FUNCTION_BLOCK ValueObjectUDINT EXTENDS ValueObject
  VAR
    lValue : UDINT := 0;
    lOverrideValue : UDINT;
  END_VAR

            
          

METHOD configure
  VAR_INPUT
    executeContext : POINTER TO ExecuteContext;
  END_VAR
                  IF (executeContext^.configureUDINT(cTokenValue,lValue,FALSE,THIS)) THEN
	RETURN;
END_IF

IF (executeContext^.configureUDINT(cTokenOverrideValue,lOverrideValue,FALSE,THIS)) THEN
	RETURN;
END_IF

SUPER^.configure(executeContext);

                
END_METHOD

METHOD describe
  VAR_INPUT
    executeContext : POINTER TO ExecuteContext;
  END_VAR
                  SUPER^.describe(executeContext);

IF (executeContext^.matchOption(cExecuteOptionSyntax)) THEN
	executeContext^.describeSyntaxConfigurable(lStyle,cTokenValue,cDataTypeUDINT,cEnumTypeNone,lUnits,cDescriptionValue);
	executeContext^.describeSyntaxConfigurable(cValueStyleParameter,cTokenOverrideValue,cDataTypeUDINT,cEnumTypeNone,lUnits,cDescriptionOverrideValue);

	RETURN;
END_IF

IF (executeContext^.matchOption(cExecuteOptionParameter)) THEN
	executeContext^.describeParameter(lStyle,lIdentity,cTokenValue,gTypeHandler.getTokenForUDINT(lValue),cDataTypeUDINT,cEnumTypeNone,lUnits,cDescriptionValue);
	executeContext^.describeParameter(cValueStyleParameter,lIdentity,cTokenOverrideValue,gTypeHandler.getTokenForUDINT(lOverrideValue),cDataTypeUDINT,cEnumTypeNone,lUnits,cDescriptionOverrideValue);
		
	RETURN;
END_IF

executeContext^.appendTokenPair(cTokenValue,gTypeHandler.getTokenForUDINT(lValue),FALSE,TRUE);
executeContext^.appendTokenPair(cTokenOverrideValue,gTypeHandler.getTokenForUDINT(lOverrideValue),FALSE,TRUE);



                
END_METHOD

METHOD operator
                  IF (lOverride) THEN
	lValue := lOverrideValue;
END_IF


                
END_METHOD

PROPERTY OverrideValue : UDINT
GET
                    OverrideValue := lOverrideValue;
                  
END_GET
SET
                    lOverrideValue := OverrideValue;
                  
END_SET
END_PROPERTY

PROPERTY TypeToken : t_medium_string
GET
                    TypeToken := 'ValObjUDINT';
                  
END_GET
END_PROPERTY

(* {attribute 'monitoring' := 'call'} *)
PROPERTY Value : UDINT
GET
                    Value := lValue;
                  
END_GET
SET
                    lValue := Value;
                  
END_SET
END_PROPERTY
END_FUNCTION_BLOCK

FUNCTION_BLOCK ValueReferenceUDINT EXTENDS ValueReference
  VAR
    lValue : REFERENCE TO UDINT;
  END_VAR

            
          

METHOD configure
  VAR_INPUT
    executeContext : POINTER TO ExecuteContext;
  END_VAR
                  IF (executeContext^.configureUDINT(cTokenValue,lValue,FALSE,THIS)) THEN
	RETURN;
END_IF

SUPER^.configure(executeContext);


                
END_METHOD

METHOD describe
  VAR_INPUT
    executeContext : POINTER TO ExecuteContext;
  END_VAR
                  IF (executeContext^.matchOption(cExecuteOptionParameter)) THEN
	executeContext^.describeParameter(lStyle,lIdentity,cTokenValue,gTypeHandler.getTokenForUDINT(lValue),cDataTypeUDINT,cEnumTypeNone,lUnits,cDescriptionValue);
	RETURN;
END_IF

SUPER^.describe(executeContext);

IF (executeContext^.matchOption(cExecuteOptionSyntax)) THEN
	executeContext^.describeSyntaxConfigurable(lStyle,cTokenValue,cDataTypeUDINT,cEnumTypeNone,lUnits,cDescriptionValue);
	RETURN;
END_IF

executeContext^.appendTokenPair(cTokenValue,gTypeHandler.getTokenForUDINT(lValue),FALSE,TRUE);





                
END_METHOD

METHOD initializeValueReference
  VAR_INPUT
    value : REFERENCE TO UDINT;
    p : POINTER TO t_particle_nop;
    _name : t_medium_string;
    description : t_long_string;
    units : t_token_string;
    style : t_value_style;
  END_VAR
                  lValue REF= value;
Name := _name;
Description := description;
lUnits := units;
lStyle := style;

IF (p<>0) THEN
	p^.registerNonOperational(THIS);
END_IF

                
END_METHOD

PROPERTY TypeToken : t_medium_string
GET
                    TypeToken := 'ValRefUDINT';
                  
END_GET
END_PROPERTY

PROPERTY Value : UDINT
GET
                    Value := lValue;
                  
END_GET
SET
                    lValue := Value;
                  
END_SET
END_PROPERTY
END_FUNCTION_BLOCK

FUNCTION_BLOCK ValueObjectUINTInputReferenceUINT EXTENDS ValueObjectUINT
  VAR
    lInputReference : REFERENCE TO UINT;
  END_VAR

            
          

METHOD initialize
                  IF (NOT(__ISVALIDREF(lInputReference))) THEN
	gCodeErrorHandler(pMessage:=CONCAT('null reference in ',lIdentity));
END_IF

SUPER^.initialize();

                
END_METHOD

METHOD operator
                  lValue := lInputReference;

SUPER^.operator();

                
END_METHOD

PROPERTY InputReference : REFERENCE TO UINT
SET
                    lInputReference REF= InputReference;


                  
END_SET
END_PROPERTY
END_FUNCTION_BLOCK

FUNCTION_BLOCK ValueObjectUINTOutputReferenceUINT EXTENDS ValueObjectUINT
  VAR
    lOutputReference : REFERENCE TO UINT;
  END_VAR

            
          

METHOD initialize
                  IF (NOT(__ISVALIDREF(lOutputReference))) THEN
	gCodeErrorHandler(pMessage:=CONCAT('null reference in ',lIdentity));
END_IF

SUPER^.initialize();

                
END_METHOD

METHOD operator
                  SUPER^.operator();

lOutputReference := lValue;
                
END_METHOD

PROPERTY OutputReference : REFERENCE TO UINT
SET
                    lOutputReference ref= OutputReference;
                  
END_SET
END_PROPERTY
END_FUNCTION_BLOCK

FUNCTION_BLOCK ValueObjectUINT EXTENDS ValueObject
  VAR
    lValue : UINT := 0;
    lOverrideValue : UINT := 0;
  END_VAR

            
          

METHOD configure
  VAR_INPUT
    executeContext : POINTER TO ExecuteContext;
  END_VAR
                  IF (executeContext^.configureUINT(cTokenValue,lValue,FALSE,THIS)) THEN
	RETURN;
END_IF

IF (executeContext^.configureUINT(cTokenOverrideValue,lOverrideValue,FALSE,THIS)) THEN
	RETURN;
END_IF

SUPER^.configure(executeContext);

                
END_METHOD

METHOD describe
  VAR_INPUT
    executeContext : POINTER TO ExecuteContext;
  END_VAR
                  SUPER^.describe(executeContext);

IF (executeContext^.matchOption(cExecuteOptionSyntax)) THEN
	executeContext^.describeSyntaxConfigurable(lStyle,cTokenValue,cDataTypeUINT,cEnumTypeNone,lUnits,cDescriptionValue);
	executeContext^.describeSyntaxConfigurable(cValueStyleParameter,cTokenOverrideValue,cDataTypeUINT,cEnumTypeNone,lUnits,cDescriptionOverrideValue);

	RETURN;
END_IF

IF (executeContext^.matchOption(cExecuteOptionParameter)) THEN
	executeContext^.describeParameter(lStyle,lIdentity,cTokenValue,gTypeHandler.getTokenForUINT(lValue),cDataTypeUINT,cEnumTypeNone,lUnits,cDescriptionValue);
	executeContext^.describeParameter(cValueStyleParameter,lIdentity,cTokenOverrideValue,gTypeHandler.getTokenForUINT(lOverrideValue),cDataTypeUINT,cEnumTypeNone,lUnits,cDescriptionOverrideValue);
		
	RETURN;
END_IF

executeContext^.appendTokenPair(cTokenValue,gTypeHandler.getTokenForUINT(lValue),FALSE,TRUE);
executeContext^.appendTokenPair(cTokenOverrideValue,gTypeHandler.getTokenForUINT(lOverrideValue),FALSE,TRUE);




                
END_METHOD

METHOD operator
                  IF (lOverride) THEN
	lValue := lOverrideValue;
END_IF

                
END_METHOD

PROPERTY OverrideValue : UINT
GET
                    OverrideValue := lOverrideValue;
                  
END_GET
SET
                    lOverrideValue := OverrideValue;
                  
END_SET
END_PROPERTY

PROPERTY TypeToken : t_medium_string
GET
                    TypeToken := 'ValObjUINT';
                  
END_GET
END_PROPERTY

PROPERTY Value : UINT
GET
                    Value := lValue;
                  
END_GET
SET
                    lValue := Value;
                  
END_SET
END_PROPERTY

PROPERTY ValueReference : REFERENCE TO UINT
GET
                    ValueReference REF= lValue;

                  
END_GET
END_PROPERTY
END_FUNCTION_BLOCK

FUNCTION_BLOCK ValueReferencePersistentUINT EXTENDS ValueReference
  VAR
    lValue : REFERENCE TO t_persistent_uint;
  END_VAR

            
          

METHOD describe
  VAR_INPUT
    executeContext : POINTER TO ExecuteContext;
  END_VAR
                  IF (executeContext^.matchOption(cExecuteOptionParameter)) THEN
	executeContext^.describeParameter(lStyle,lIdentity,cTokenValue,gTypeHandler.getTokenForUINT(lValue.Value),cDataTypeUINT,cEnumTypeNone,lUnits,cDescriptionValue);	
	RETURN;
END_IF

SUPER^.describe(executeContext);

IF (executeContext^.matchOption(cExecuteOptionSyntax)) THEN
	executeContext^.describeSyntaxConfigurable(lStyle,cTokenValue,cDataTypeUINT,cEnumTypeNone,lUnits,cDescriptionValue);
	RETURN;
END_IF

executeContext^.appendTokenPair(cTokenValue,gTypeHandler.getTokenForUINT(lValue.Value),FALSE,TRUE);

                
END_METHOD

METHOD configure
  VAR_INPUT
    executeContext : POINTER TO ExecuteContext;
  END_VAR
  VAR
    value : UINT;
  END_VAR
                  IF (executeContext^.configureUINT(cTokenValue,value,FALSE,THIS)) THEN
	lValue.Value := value;
	RETURN;
END_IF

SUPER^.configure(executeContext);

                
END_METHOD

METHOD initializeValueReference
  VAR_INPUT
    value : REFERENCE TO t_persistent_uint;
    p : POINTER TO t_particle_nop;
    _name : t_medium_string;
    description : t_long_string;
    units : t_token_string;
    style : t_value_style;
  END_VAR
                  lValue REF= value;
Name := _name;
Description := description;
lUnits := units;
lStyle := style;

IF (p<>0) THEN
	p^.registerNonOperational(THIS);
END_IF

                
END_METHOD

PROPERTY TypeToken : t_medium_string
GET
                    TypeToken := 'ValRefPersUINT';
                  
END_GET
END_PROPERTY

PROPERTY Value : UINT
GET
                    Value := lValue.Value;
                  
END_GET
SET
                    lValue.Value := Value;
                  
END_SET
END_PROPERTY
END_FUNCTION_BLOCK

FUNCTION_BLOCK ValueReferenceUINT EXTENDS ValueReference
  VAR
    lValue : REFERENCE TO UINT;
  END_VAR

            
          

METHOD configure
  VAR_INPUT
    executeContext : POINTER TO ExecuteContext;
  END_VAR
                  IF (executeContext^.configureUINT(cTokenValue,lValue,FALSE,THIS)) THEN
	RETURN;
END_IF

SUPER^.configure(executeContext);


                
END_METHOD

METHOD initializeValueReference
  VAR_INPUT
    value : REFERENCE TO UINT;
    p : POINTER TO t_particle_nop;
    _name : t_medium_string;
    description : t_long_string;
    units : t_token_string;
    style : t_value_style;
  END_VAR
                  lValue REF= value;
Name := _name;
Description := description;
lUnits := units;
lStyle := style;

IF (p<>0) THEN
	p^.registerNonOperational(THIS);
END_IF

                
END_METHOD

METHOD describe
  VAR_INPUT
    executeContext : POINTER TO ExecuteContext;
  END_VAR
                  IF (executeContext^.matchOption(cExecuteOptionParameter)) THEN
	executeContext^.describeParameter(lStyle,lIdentity,cTokenValue,gTypeHandler.getTokenForUINT(lValue),cDataTypeUINT,cEnumTypeNone,lUnits,cDescriptionValue);
	RETURN;
END_IF

SUPER^.describe(executeContext);

IF (executeContext^.matchOption(cExecuteOptionSyntax)) THEN
	executeContext^.describeSyntaxConfigurable(lStyle,cTokenValue,cDataTypeUINT,cEnumTypeNone,lUnits,cDescriptionValue);
	RETURN;
END_IF

executeContext^.appendTokenPair(cTokenValue,gTypeHandler.getTokenForUINT(lValue),FALSE,TRUE);



                
END_METHOD

PROPERTY TypeToken : t_medium_string
GET
                    TypeToken := 'ValRefUINT';
                  
END_GET
END_PROPERTY

PROPERTY Value : UINT
GET
                    Value := lValue;
                  
END_GET
SET
                    lValue := Value;
                  
END_SET
END_PROPERTY
END_FUNCTION_BLOCK

FUNCTION_BLOCK ValueObjectULINTInputReferenceULINT EXTENDS ValueObjectULINT
  VAR
    lInputReference : REFERENCE TO ULINT;
  END_VAR

            
          

METHOD initialize
                  IF (NOT(__ISVALIDREF(lInputReference))) THEN
	gCodeErrorHandler(pMessage:=CONCAT('null reference in ',lIdentity));
END_IF

SUPER^.initialize();

                
END_METHOD

METHOD operator
                  lValue := lInputReference;

SUPER^.operator();

                
END_METHOD

PROPERTY InputReference : REFERENCE TO ULINT
SET
                    lInputReference REF= InputReference;


                  
END_SET
END_PROPERTY
END_FUNCTION_BLOCK

FUNCTION_BLOCK ValueObjectULINT EXTENDS ValueObject
  VAR
    lValue : ULINT := 0;
    lOverrideValue : ULINT;
  END_VAR

            
          

METHOD configure
  VAR_INPUT
    executeContext : POINTER TO ExecuteContext;
  END_VAR
                  IF (executeContext^.configureULINT(cTokenValue,lValue,FALSE,THIS)) THEN
	RETURN;
END_IF

IF (executeContext^.configureULINT(cTokenOverrideValue,lOverrideValue,FALSE,THIS)) THEN
	RETURN;
END_IF

SUPER^.configure(executeContext);


                
END_METHOD

METHOD describe
  VAR_INPUT
    executeContext : POINTER TO ExecuteContext;
  END_VAR
                  SUPER^.describe(executeContext);

IF (executeContext^.matchOption(cExecuteOptionSyntax)) THEN
	executeContext^.describeSyntaxConfigurable(lStyle,cTokenValue,cDataTypeULINT,cEnumTypeNone,lUnits,cDescriptionValue);
	executeContext^.describeSyntaxConfigurable(cValueStyleParameter,cTokenOverrideValue,cDataTypeULINT,cEnumTypeNone,lUnits,cDescriptionOverrideValue);
	
	RETURN;
END_IF

IF (executeContext^.matchOption(cExecuteOptionParameter)) THEN
	executeContext^.describeParameter(lStyle,lIdentity,cTokenValue,gTypeHandler.getTokenForULINT(lValue),cDataTypeULINT,cEnumTypeNone,lUnits,cDescriptionValue);
	executeContext^.describeParameter(cValueStyleParameter,lIdentity,cTokenOverrideValue,gTypeHandler.getTokenForULINT(lOverrideValue),cDataTypeULINT,cEnumTypeNone,lUnits,cDescriptionOverrideValue);
		
	RETURN;
END_IF

executeContext^.appendTokenPair(cTokenValue,gTypeHandler.getTokenForULINT(lValue),FALSE,TRUE);
executeContext^.appendTokenPair(cTokenOverrideValue,gTypeHandler.getTokenForULINT(lOverrideValue),FALSE,TRUE);



                
END_METHOD

METHOD operator
                  IF (lOverride) THEN
	lValue := lOverrideValue;
END_IF


                
END_METHOD

PROPERTY OverrideValue : ULINT
GET
                    OverrideValue := lOverrideValue;
                  
END_GET
SET
                    lOverrideValue := OverrideValue;
                  
END_SET
END_PROPERTY

PROPERTY TypeToken : t_medium_string
GET
                    TypeToken := 'ValObjULINT';
                  
END_GET
END_PROPERTY

PROPERTY Value : ULINT
GET
                    Value := lValue;
                  
END_GET
SET
                    lValue := Value;
                  
END_SET
END_PROPERTY
END_FUNCTION_BLOCK

FUNCTION_BLOCK ValueReferenceULINT EXTENDS ValueReference
  VAR
    lValue : REFERENCE TO ULINT;
  END_VAR

            
          

METHOD configure
  VAR_INPUT
    executeContext : POINTER TO ExecuteContext;
  END_VAR
                  IF (executeContext^.configureULINT(cTokenValue,lValue,FALSE,THIS)) THEN
	RETURN;
END_IF

SUPER^.configure(executeContext);



                
END_METHOD

METHOD describe
  VAR_INPUT
    executeContext : POINTER TO ExecuteContext;
  END_VAR
                  IF (executeContext^.matchOption(cExecuteOptionParameter)) THEN
	executeContext^.describeParameter(lStyle,lIdentity,cTokenValue,gTypeHandler.getTokenForULINT(lValue),cDataTypeULINT,cEnumTypeNone,lUnits,cDescriptionValue);
	RETURN;
END_IF

SUPER^.describe(executeContext);

IF (executeContext^.matchOption(cExecuteOptionSyntax)) THEN
	executeContext^.describeSyntaxConfigurable(lStyle,cTokenValue,cDataTypeULINT,cEnumTypeNone,lUnits,cDescriptionValue);
	RETURN;
END_IF

executeContext^.appendTokenPair(cTokenValue,gTypeHandler.getTokenForULINT(lValue),FALSE,TRUE);



                
END_METHOD

METHOD initializeValueReference
  VAR_INPUT
    value : REFERENCE TO ULINT;
    p : POINTER TO t_particle_nop;
    _name : t_medium_string;
    description : t_long_string;
    units : t_token_string;
    style : t_value_style;
  END_VAR
                  lValue REF= value;
Name := _name;
Description := description;
lUnits := units;
lStyle := style;

IF (p<>0) THEN
	p^.registerNonOperational(THIS);
END_IF

                
END_METHOD

PROPERTY TypeToken : t_medium_string
GET
                    TypeToken := 'ValRefULINT';
                  
END_GET
END_PROPERTY

PROPERTY Value : ULINT
GET
                    Value := lValue;
                  
END_GET
SET
                    lValue := Value;
                  
END_SET
END_PROPERTY
END_FUNCTION_BLOCK

FUNCTION_BLOCK ValueObjectUSINTInputReferenceUSINT EXTENDS ValueObjectUSINT
  VAR
    lInputReference : REFERENCE TO USINT;
  END_VAR

            
          

METHOD initialize
                  IF (NOT(__ISVALIDREF(lInputReference))) THEN
	gCodeErrorHandler(pMessage:=CONCAT('null reference in ',lIdentity));
END_IF

SUPER^.initialize();

                
END_METHOD

METHOD operator
                  lValue := lInputReference;

SUPER^.operator();

                
END_METHOD

PROPERTY InputReference : REFERENCE TO USINT
SET
                    lInputReference REF= InputReference;


                  
END_SET
END_PROPERTY
END_FUNCTION_BLOCK

FUNCTION_BLOCK ValueObjectUSINTInputUSINT EXTENDS ValueObjectUSINT
  VAR
    lInput : USINT;
  END_VAR

            
          

METHOD operator
                  lValue := lInput;

SUPER^.operator();

                
END_METHOD

PROPERTY Input : USINT
SET
                    lInput := Input;
operator();

                  
END_SET
END_PROPERTY
END_FUNCTION_BLOCK

FUNCTION_BLOCK ValueObjectUSINTOutputReferenceUSINT EXTENDS ValueObjectUSINT
  VAR
    lOutputReference : REFERENCE TO USINT;
  END_VAR

            
          

METHOD initialize
                  IF (NOT(__ISVALIDREF(lOutputReference))) THEN
	gCodeErrorHandler(pMessage:=CONCAT('null reference in ',lIdentity));
END_IF

SUPER^.initialize();

                
END_METHOD

METHOD operator
                  SUPER^.operator();

lOutputReference := lValue;

                
END_METHOD

PROPERTY OutputReference : REFERENCE TO USINT
SET
                    lOutputReference ref= OutputReference;
                  
END_SET
END_PROPERTY
END_FUNCTION_BLOCK

FUNCTION_BLOCK ValueObjectUSINT EXTENDS ValueObject
  VAR
    lValue : USINT := 0;
    lOverrideValue : USINT := 0;
  END_VAR

            
          

METHOD configure
  VAR_INPUT
    executeContext : POINTER TO ExecuteContext;
  END_VAR
                  IF (executeContext^.configureUSINT(cTokenValue,lValue,FALSE,THIS)) THEN
	RETURN;
END_IF

IF (executeContext^.configureUSINT(cTokenOverrideValue,lOverrideValue,FALSE,THIS)) THEN
	RETURN;
END_IF

SUPER^.configure(executeContext);

                
END_METHOD

METHOD describe
  VAR_INPUT
    executeContext : POINTER TO ExecuteContext;
  END_VAR
                  SUPER^.describe(executeContext);

IF (executeContext^.matchOption(cExecuteOptionSyntax)) THEN
	executeContext^.describeSyntaxConfigurable(lStyle,cTokenValue,cDataTypeUSINT,cEnumTypeNone,lUnits,cDescriptionValue);
	executeContext^.describeSyntaxConfigurable(cValueStyleParameter,cTokenOverrideValue,cDataTypeUSINT,cEnumTypeNone,lUnits,cDescriptionOverrideValue);

	RETURN;
END_IF

IF (executeContext^.matchOption(cExecuteOptionParameter)) THEN
	executeContext^.describeParameter(lStyle,lIdentity,cTokenValue,gTypeHandler.getTokenForUSINT(lValue),cDataTypeUSINT,cEnumTypeNone,lUnits,cDescriptionValue);
	executeContext^.describeParameter(cValueStyleParameter,lIdentity,cTokenOverrideValue,gTypeHandler.getTokenForUSINT(lOverrideValue),cDataTypeUSINT,cEnumTypeNone,lUnits,cDescriptionOverrideValue);
	
	RETURN;
END_IF

executeContext^.appendTokenPair(cTokenValue,gTypeHandler.getTokenForUSINT(lValue),FALSE,TRUE);
executeContext^.appendTokenPair(cTokenOverrideValue,gTypeHandler.getTokenForUSINT(lOverrideValue),FALSE,TRUE);

                
END_METHOD

METHOD operator
                  IF (lOverride) THEN
	lValue := lOverrideValue;
END_IF


                
END_METHOD

PROPERTY OverrideValue : USINT
GET
                    OverrideValue := lOverrideValue;
                  
END_GET
SET
                    lOverrideValue := OverrideValue;
                  
END_SET
END_PROPERTY

PROPERTY TypeToken : t_medium_string
GET
                    TypeToken := 'ValObjUSINT';
                  
END_GET
END_PROPERTY

(* {attribute 'monitoring' := 'call'} *)
PROPERTY Value : USINT
GET
                    Value := lValue;
                  
END_GET
SET
                    lValue := Value;
                  
END_SET
END_PROPERTY
END_FUNCTION_BLOCK

FUNCTION_BLOCK ValueReferenceUSINT EXTENDS ValueReference
  VAR
    lValue : REFERENCE TO USINT;
  END_VAR

            
          

METHOD configure
  VAR_INPUT
    executeContext : POINTER TO ExecuteContext;
  END_VAR
                  IF (executeContext^.configureUSINT(cTokenValue,lValue,FALSE,THIS)) THEN
	RETURN;
END_IF

SUPER^.configure(executeContext);

                
END_METHOD

METHOD describe
  VAR_INPUT
    executeContext : POINTER TO ExecuteContext;
  END_VAR
                  IF (executeContext^.matchOption(cExecuteOptionParameter)) THEN
	executeContext^.describeParameter(lStyle,lIdentity,cTokenValue,gTypeHandler.getTokenForUSINT(lValue),cDataTypeUSINT,cEnumTypeNone,lUnits,cDescriptionValue);
	RETURN;
END_IF

SUPER^.describe(executeContext);

IF (executeContext^.matchOption(cExecuteOptionSyntax)) THEN
	executeContext^.describeSyntaxConfigurable(lStyle,cTokenValue,cDataTypeUSINT,cEnumTypeNone,lUnits,cDescriptionValue);
	RETURN;
END_IF

executeContext^.appendTokenPair(cTokenValue,gTypeHandler.getTokenForUSINT(lValue),FALSE,TRUE);



                
END_METHOD

METHOD initializeValueReference
  VAR_INPUT
    value : REFERENCE TO USINT;
    p : POINTER TO t_particle_nop;
    _name : t_medium_string;
    description : t_long_string;
    units : t_token_string;
    style : t_value_style;
  END_VAR
                  lValue REF= value;
Name := _name;
Description := description;
lUnits := units;
lStyle := style;

IF (p<>0) THEN
	p^.registerNonOperational(THIS);
END_IF

                
END_METHOD

PROPERTY TypeToken : t_medium_string
GET
                    TypeToken := 'ValRefUSINT';
                  
END_GET
END_PROPERTY

PROPERTY Value : USINT
GET
                    Value := lValue;
                  
END_GET
SET
                    lValue := Value;
                  
END_SET
END_PROPERTY
END_FUNCTION_BLOCK

FUNCTION_BLOCK ValueObject EXTENDS Particle
  VAR
    lUnits : t_token_string;
    lOverride : BOOL := FALSE;
    lStyle : t_value_style := cValueStyleConfigurable;
  END_VAR

            
          

METHOD describe
  VAR_INPUT
    executeContext : POINTER TO ExecuteContext;
  END_VAR
                  SUPER^.describe(executeContext);

IF (executeContext^.matchOption(cExecuteOptionSyntax)) THEN
	executeContext^.describeSyntaxConfigurable(cValueStyleParameter,cTokenOverride,cDataTypeBool,cEnumTypeNone,lUnits,cDescriptionOverride);
	RETURN;
END_IF

IF (executeContext^.matchOption(cExecuteOptionParameter)) THEN
	executeContext^.describeParameter(cValueStyleParameter,lIdentity,cTokenOverride,gTypeHandler.getTokenForBool(lOverride),cDataTypeBool,cEnumTypeNone,lUnits,cDescriptionOverride);

	RETURN;
END_IF

executeContext^.appendTokenPair(cTokenOverride,gTypeHandler.getTokenForUSINT(BOOL_TO_USINT(lOverride)),FALSE,TRUE);


                
END_METHOD

METHOD initializeValueObject
  VAR_INPUT
    p : POINTER TO t_particle_nop;
    _name : t_medium_string;
    description : t_long_string;
    units : t_token_string;
    style : t_value_style;
  END_VAR
                  Name := _name;
Description := description;
lUnits := units;
lStyle := style;

IF (p=0) THEN
	gCodeErrorHandler(pMessage:='initializing value with null t_particle_nop');
	RETURN;
END_IF

p^.registerNonOperational(THIS);

                
END_METHOD

METHOD initializeValueObjectOp
  VAR_INPUT
    p : POINTER TO t_particle_op;
    _name : t_medium_string;
    description : t_long_string;
    units : t_token_string;
    style : t_value_style;
  END_VAR
                  Name := _name;
Description := description;
lUnits := units;
lStyle := style;

IF (p=0) THEN
	gCodeErrorHandler(pMessage:='initializing value with null t_particle_op');
	RETURN;
END_IF

p^.registerOperational(THIS);

                
END_METHOD

METHOD configure
  VAR_INPUT
    executeContext : POINTER TO ExecuteContext;
  END_VAR
                  IF (executeContext^.configureBool(cTokenOverride,lOverride,FALSE,THIS)) THEN
	RETURN;
END_IF

SUPER^.configure(executeContext);

                
END_METHOD

PROPERTY Override : BOOL
GET
                    Override := lOverride;
                  
END_GET
SET
                    lOverride := Override;
                  
END_SET
END_PROPERTY

PROPERTY TypeToken : t_medium_string
GET
                    TypeToken := 'ValueObject';
                  
END_GET
END_PROPERTY
END_FUNCTION_BLOCK

FUNCTION_BLOCK ValueReference EXTENDS Particle
  VAR
    lUnits : t_token_string;
    lStyle : t_value_style := cValueStyleConfigurable;
  END_VAR

            
          

PROPERTY TypeToken : t_medium_string
GET
                    TypeToken := 'ValueReference';
                  
END_GET
END_PROPERTY
END_FUNCTION_BLOCK

FUNCTION_BLOCK ExecuteCommand
  VAR
    lCommand : t_token_type;
    lOptions : t_options_list;
    lPairs : ARRAY[1..4] OF t_argument;
  END_VAR

            
          
END_FUNCTION_BLOCK

{attribute 'enable_dynamic_creation'}
FUNCTION_BLOCK ExecuteContext
  VAR CONSTANT
    cExecuteLimit : USINT := 2;
    cExecutionQueueMax : UINT := 4096;
    cParseMaxTokens : USINT := 32;
    cSkipCount : USINT := 5;
  END_VAR
  VAR
    lExecutionQueue : ARRAY[1..cExecutionQueueMax] OF t_execution_queue_item;  (* lSource: REFERENCE TO t_execute_source; *)
    lExecutionQueueCount : UINT;
    lExecutionQueueIndex : UINT;
    lRegisterDepth : USINT;
    lCurrentCommand : t_command_request;
    lExecuteReturn : t_execute_return := cExecuteReturnOK;
    lResponsePending : BOOL := FALSE;
    lError : BOOL := FALSE;
    lReportError : BOOL := FALSE;
    lWriteStream : t_stream;
    lEnableExecutor : BOOL := TRUE;
    lReadWrite : BOOL := FALSE;
    lPassCount : USINT;
    lPassLimit : USINT := cExecuteLimit;
    lSkipIndex : USINT := 0;
    lSkipCount : USINT := cSkipCount;
    lCommaPending : BOOL := FALSE;
    lWrappedResponse : BOOL := FALSE;
  END_VAR

            
          

METHOD configureDWORD : BOOL
  VAR_INPUT
    parameter : t_token_type;
    target : REFERENCE TO DWORD;
    required : BOOL;
    particle : POINTER TO t_particle;
  END_VAR
  VAR
    valueToken : t_token_string;
  END_VAR
                  configureDWORD := matchArgument(parameter,valueToken);

IF (NOT(configureDWORD)) THEN
	IF (required) THEN
		executeContextFail(THIS,cExecuteReturnMissingArgument,TRUE);		
	END_IF
	
	RETURN;
END_IF

IF (NOT(gTypeHandler.getDWORDFromToken(valueToken,target))) THEN
	executeContextFail(THIS,cExecuteReturnParseParameterError,TRUE);
	RETURN;
END_IF

gSystemServices.Executor.reportParameterUpdates(particle);

                
END_METHOD

METHOD describeSyntaxConfigurable
  VAR_INPUT
    style : t_value_style;
    parameter : t_token_type;
    dataType : t_data_type;
    enumType : t_enum_type;
    units : t_token_string;
    description : REFERENCE TO t_long_string;
  END_VAR
                  recordInitiator();

appendTokenPair(parameter,gTypeHandler.getTokenForDataType(dataType),TRUE,FALSE);

append(', "_metadata":');
recordInitiator();

appendPair('style',gTypeHandler.getTokenForEnum(cEnumTypeValueStyle,style),TRUE,FALSE);
appendPair('units',units,TRUE,TRUE);
appendPair('description',description,TRUE,TRUE);

IF (enumType<>cEnumTypeNone) THEN
	appendPair('enum',gTypeHandler.getStringForEnumOptions(enumType),FALSE,TRUE);
END_IF

recordTerminator();
recordTerminatorWithNewline();

                
END_METHOD

METHOD configureUSINT : BOOL
  VAR_INPUT
    parameter : t_token_type;
    target : REFERENCE TO USINT;
    required : BOOL;
    particle : POINTER TO t_particle;
  END_VAR
  VAR
    valueToken : t_token_string;
  END_VAR
                  configureUSINT := matchArgument(parameter,valueToken);

IF (NOT(configureUSINT)) THEN
	IF (required) THEN
		executeContextFail(THIS,cExecuteReturnMissingArgument,TRUE);		
	END_IF
	
	RETURN;
END_IF

IF (NOT(gTypeHandler.getUSINTFromToken(valueToken,target))) THEN
	executeContextFail(THIS,cExecuteReturnParseParameterError,TRUE);
	RETURN;
END_IF

gSystemServices.Executor.reportParameterUpdates(particle);

                
END_METHOD

METHOD recordInitiatorWithNewlineIndent
                  formatWithNewlineIndent();
lWriteStream.recordInitiator();

                
END_METHOD

METHOD formatWithNewlineIndent
                  IF (NOT(lWrappedResponse)) THEN
	lWriteStream.newline();
	lWriteStream.indent();
END_IF


                
END_METHOD

METHOD append
  VAR_INPUT
    str : STRING;
  END_VAR
                  lWriteStream.append(str);

                
END_METHOD

METHOD configureUINT : BOOL
  VAR_INPUT
    parameter : t_token_type;
    target : REFERENCE TO UINT;
    required : BOOL;
    particle : POINTER TO t_particle;
  END_VAR
  VAR
    valueToken : t_token_string;
  END_VAR
                  configureUINT := matchArgument(parameter,valueToken);

IF (NOT(configureUINT)) THEN
	IF (required) THEN
		executeContextFail(THIS,cExecuteReturnMissingArgument,TRUE);		
	END_IF
	
	RETURN;
END_IF

IF (NOT(gTypeHandler.getUINTFromToken(valueToken,target))) THEN
	executeContextFail(THIS,cExecuteReturnParseParameterError,TRUE);
	RETURN;
END_IF

gSystemServices.Executor.reportParameterUpdates(particle);

                
END_METHOD

METHOD configureMediumString : BOOL
  VAR_INPUT
    parameter : t_token_type;
    target : REFERENCE TO t_medium_string;
    required : BOOL;
    particle : POINTER TO t_particle;
  END_VAR
  VAR
    valueToken : t_token_string;
  END_VAR
                  configureMediumString := matchArgument(parameter,valueToken);

IF (NOT(configureMediumString)) THEN
	IF (required) THEN
		executeContextFail(THIS,cExecuteReturnMissingArgument,TRUE);		
	END_IF
	
	RETURN;
END_IF

target := valueToken;

gSystemServices.Executor.reportParameterUpdates(particle);

                
END_METHOD

METHOD configureUDINT : BOOL
  VAR_INPUT
    parameter : t_token_type;
    target : REFERENCE TO UDINT;
    required : BOOL;
    particle : POINTER TO t_particle;
  END_VAR
  VAR
    valueToken : t_token_string;
  END_VAR
                  configureUDINT := matchArgument(parameter,valueToken);

IF (NOT(configureUDINT)) THEN
	IF (required) THEN
		executeContextFail(THIS,cExecuteReturnMissingArgument,TRUE);		
	END_IF
	
	RETURN;
END_IF

IF (NOT(gTypeHandler.getUDINTFromToken(valueToken,target))) THEN
	executeContextFail(THIS,cExecuteReturnParseParameterError,TRUE);
	RETURN;
END_IF

gSystemServices.Executor.reportParameterUpdates(particle);


                
END_METHOD

METHOD configureReal : BOOL
  VAR_INPUT
    parameter : t_token_type;
    target : REFERENCE TO REAL;
    required : BOOL;
    particle : POINTER TO t_particle;
  END_VAR
  VAR
    valueToken : t_token_string;
  END_VAR
                  configureReal := matchArgument(parameter,valueToken);

IF (NOT(configureReal)) THEN
	IF (required) THEN
		executeContextFail(THIS,cExecuteReturnMissingArgument,TRUE);		
	END_IF
	
	RETURN;
END_IF

IF (NOT(gTypeHandler.getREALFromToken(valueToken,target))) THEN
	executeContextFail(THIS,cExecuteReturnParseParameterError,TRUE);
	RETURN;
END_IF

gSystemServices.Executor.reportParameterUpdates(particle);


                
END_METHOD

METHOD configurePercentage : BOOL
  VAR_INPUT
    parameter : t_token_type;
    target : REFERENCE TO t_percentage;
    required : BOOL;
    particle : POINTER TO t_particle;
  END_VAR
  VAR
    valueToken : t_token_string;
  END_VAR
                  configurePercentage := matchArgument(parameter,valueToken);

IF (NOT(configurePercentage)) THEN
	IF (required) THEN
		executeContextFail(THIS,cExecuteReturnMissingArgument,TRUE);		
	END_IF
	
	RETURN;
END_IF

IF (NOT(gTypeHandler.getPercentageFromToken(valueToken,target))) THEN
	executeContextFail(THIS,cExecuteReturnParseParameterError,TRUE);
	RETURN;
END_IF

gSystemServices.Executor.reportParameterUpdates(particle);


                
END_METHOD

METHOD configureEnum : BOOL
  VAR_INPUT
    enumType : t_enum_type;
    parameter : t_token_type;
    target : REFERENCE TO INT;
    required : BOOL;
    particle : POINTER TO t_particle;
  END_VAR
  VAR
    valueToken : t_token_string;
  END_VAR
                  configureEnum := matchArgument(parameter,valueToken);

IF (NOT(configureEnum)) THEN
	IF (required) THEN
		executeContextFail(THIS,cExecuteReturnMissingArgument,TRUE);		
	END_IF
	
	RETURN;
END_IF

IF (NOT(gTypeHandler.getEnumFromToken(enumType,valueToken,target))) THEN
	executeContextFail(THIS,cExecuteReturnParseParameterError,TRUE);
	RETURN;
END_IF

gSystemServices.Executor.reportParameterUpdates(particle);


                
END_METHOD

METHOD configureULINT : BOOL
  VAR_INPUT
    parameter : t_token_type;
    target : REFERENCE TO ULINT;
    required : BOOL;
    particle : POINTER TO t_particle;
  END_VAR
  VAR
    valueToken : t_token_string;
  END_VAR
                  configureULINT := matchArgument(parameter,valueToken);

IF (NOT(configureULINT)) THEN
	IF (required) THEN
		executeContextFail(THIS,cExecuteReturnMissingArgument,TRUE);		
	END_IF
	
	RETURN;
END_IF

IF (NOT(gTypeHandler.getULINTFromToken(valueToken,target))) THEN
	executeContextFail(THIS,cExecuteReturnParseParameterError,TRUE);
	RETURN;
END_IF

gSystemServices.Executor.reportParameterUpdates(particle);


                
END_METHOD

METHOD operator
  VAR
    i : USINT;
  END_VAR
                  lPassCount := 0;
lWriteStream.clear();

IF (lSkipIndex<lSkipCount) THEN
	lSkipIndex := lSkipIndex + 1;
	RETURN;
END_IF
lSkipIndex := 0;

WHILE (NOT(PassComplete)) DO
	IF (ExecutionComplete) THEN
		
		IF (lResponsePending) THEN
			lResponsePending := FALSE;

			IF (lWrappedResponse) THEN
				append('], '); 
				lCommaPending := FALSE;

				appendPair('return',gTypeHandler.getTokenForEnum(cEnumTypeExecuteReturn,lExecuteReturn),TRUE,FALSE);	
				lWriteStream.recordTerminatorWithNewline();
				RETURN;
			END_IF

			IF ((lReportError) AND
				(NOT(lExecuteReturn=cExecuteReturnOK))) THEN
				append(gTypeHandler.getTokenForEnum(cEnumTypeExecuteReturn,lExecuteReturn));
				lWriteStream.newline();
			END_IF
		END_IF
		
		IF (NOT(getNextExecuteCommand())) THEN
			RETURN;
		END_IF
		
		IF (NOT(lResponsePending)) THEN
			lResponsePending := TRUE;

			IF (lWrappedResponse) THEN
				lCommaPending := FALSE;
				recordInitiator();
				append('"response": [');
			END_IF
		END_IF
	END_IF

	executeNextInQueue();
END_WHILE

                
END_METHOD

METHOD describeVerify
  VAR_INPUT
    identity : t_long_string;
    status : BOOL;
    message : t_long_string;
  END_VAR
                  lWriteStream.recordInitiator();	

lWriteStream.appendPair('identity',identity,TRUE,FALSE);
lWriteStream.appendPair('message',message,TRUE,TRUE);
lWriteStream.appendPair('status',gTypeHandler.getTokenForBool(status),FALSE,TRUE);

lWriteStream.recordTerminatorWithNewline();	

ExecuteReturn := cExecuteReturnOKNOK;
                
END_METHOD

METHOD registerExecution : BOOL
  VAR_INPUT
    particle : t_particle_ptr;
  END_VAR
                  IF (particle=0) THEN
	ExecuteReturn := cExecuteReturnExecutionQueueNullParticle;
	lError := TRUE;
	
	RETURN;
END_IF

particle^.recurse(THIS);

// eolus := getUDINTFromToken(executeContext^.ParameterToken,index,lParseOK);


                
END_METHOD

METHOD registerParticle
  VAR_INPUT
    particle : t_particle_ptr;
  END_VAR
                  IF (lExecutionQueueCount>=cExecutionQueueMax) THEN
	executeContextFail(THIS,cExecuteReturnExecutionQueueOverflow,TRUE);
	RETURN;
END_IF

IF (particle=0) THEN
	executeContextFail(THIS,cExecuteReturnExecutionQueueNullParticle,TRUE);
	RETURN;
END_IF

lExecutionQueueCount := lExecutionQueueCount + 1;

lExecutionQueue[lExecutionQueueCount].depth := lRegisterDepth;
lExecutionQueue[lExecutionQueueCount].particle := particle;

                
END_METHOD

METHOD executeNextInQueue
  VAR
    i : USINT;
    iterations : USINT;
  END_VAR
                  IF (ExecutionComplete) THEN
	RETURN;
END_IF

IF (PassComplete) THEN
	RETURN;
END_IF

lExecutionQueueIndex := lExecutionQueueIndex + 1;
lPassCount := lPassCount + 1;

FOR i:=1 TO lCurrentCommand.argumentCount DO
	lCurrentCommand.arguments[i].processed := FALSE;
END_FOR

iterations := 0;
WHILE ((NOT(Error)) AND
	(((lCurrentCommand.command=cTokenConfigure) AND (ArgsUnprocessed)) OR
	(iterations=0))) DO	
	
	lExecutionQueue[lExecutionQueueIndex].particle^.execute(THIS);
	
	IF (iterations>lCurrentCommand.argumentCount) THEN
		executeContextFail(THIS,cExecuteReturnInternalError,TRUE);
	END_IF
	iterations := iterations + 1;
	
END_WHILE

IF (ArgsUnprocessed) THEN
	executeContextFail(THIS,cExecuteReturnUnprocessedArguments,TRUE);
END_IF

IF (matchOption(cExecuteOptionPersist)) THEN
	IF (NOT(gSystemServices.PLC.persistCommand(lCurrentCommand))) THEN
		executeContextFail(THIS,cExecuteReturnPersistFailed,TRUE);
	END_IF
END_IF

                
END_METHOD

METHOD registerDepthIncrease
                  IF (lRegisterDepth<255) THEN
	lRegisterDepth := lRegisterDepth + 1;
END_IF

                
END_METHOD

METHOD registerDepthDecrease
                  IF (lRegisterDepth>0) THEN
	lRegisterDepth := lRegisterDepth - 1;
END_IF

                
END_METHOD

METHOD describeSyntaxExecutable
  VAR_INPUT
    command : REFERENCE TO t_command_definition;
  END_VAR
  VAR
    options : t_long_string;
    str : t_long_string;
    i : USINT;
  END_VAR
                  recordInitiator();

appendPair('command',gTypeHandler.getTokenForEnum(cEnumTypeTokenType,command.command),TRUE,FALSE);

append(', "_metadata":');
recordInitiator();

options := '[';

FOR i:=1 TO command.optionCount DO
	IF (i=1) THEN
		options := CONCAT(options,'"');
	ELSE
		options := CONCAT(options,', "');
	END_IF

	options := CONCAT(options,gTypeHandler.getTokenForEnum(cEnumTypeExecuteOption,command.options[i]));
	options := CONCAT(options,'"');
END_FOR

options := CONCAT(options,']');

appendPair('options',options,TRUE,FALSE);
IF (__ISVALIDREF(command.description)) THEN
	appendPair('description',command.description,TRUE,TRUE);
END_IF

recordTerminator();
recordTerminatorWithNewline();

                
END_METHOD

METHOD appendPair
  VAR_INPUT
    parameter : STRING;
    value : STRING;
    quoted : BOOL;
    comma : BOOL;
  END_VAR
  VAR
    stmp : STRING;
  END_VAR
                  IF (strcmp(value,'')) THEN
	RETURN;
END_IF

lWriteStream.appendPair(parameter,value,quoted,comma);



                
END_METHOD

METHOD recordInitiator
                  IF ((lWrappedResponse) AND (lCommaPending)) THEN
	lWriteStream.append(', ');
	lCommaPending := FALSE;
END_IF

lWriteStream.recordInitiator();

                
END_METHOD

METHOD recordTerminator
                  lWriteStream.recordTerminator();

                
END_METHOD

METHOD recordTerminatorWithNewline
                  IF (lWrappedResponse) THEN
	lWriteStream.recordTerminator();
	lCommaPending := TRUE;
	
	RETURN;
END_IF

lWriteStream.recordTerminatorWithNewline();

                
END_METHOD

METHOD describeParameter
  VAR_INPUT
    style : t_value_style;
    identity : t_long_string;
    parameter : t_token_type;
    value : t_medium_string;
    dataType : t_data_type;
    enumType : t_enum_type;
    units : t_token_string;
    description : REFERENCE TO t_long_string;
  END_VAR
  VAR
    id : t_long_string;
    quoted : BOOL;
  END_VAR
                  IF (style<>cValueStyleParameter) THEN
	RETURN;
END_IF

CASE dataType OF	
	cDataTypeNone:
		RETURN;
		
	cDataTypeEnum,
	cDataTypeString:
		quoted := TRUE;

	cDataTypeUSINT,
	cDataTypeUINT,
	cDataTypeULINT,
	cDataTypeUDINT,
	cDataTypeINT,
	cDataTypePercentage,
	cDataTypeReal,
	cDataTypeDWORD,
	cDataTypeBool:
		quoted := FALSE;
END_CASE

recordInitiator();

id := identity;
IF (parameter<>cTokenNone) THEN
	id := CONCAT(id,'/');
	id := CONCAT(id,gTypeHandler.getTokenForEnum(cEnumTypeTokenType,parameter));
END_IF

appendPair('identity',id,TRUE,FALSE);
appendPair('value',value,quoted,TRUE);

IF (NOT(matchOption(cExecuteOptionMetadata))) THEN
	recordTerminatorWithNewline();
	RETURN;
END_IF

append(', "_metadata":');
recordInitiator();

IF (enumType=cEnumTypeNone) THEN
	appendPair('type',gTypeHandler.getTokenForDataType(dataType),TRUE,FALSE);
ELSE
	appendPair('type',gTypeHandler.getTokenForEnumType(enumType),TRUE,FALSE);	
	appendPair('enum',gTypeHandler.getStringForEnumOptions(enumType),FALSE,TRUE);
END_IF

appendPair('units',units,TRUE,TRUE);
appendPair('description',description,TRUE,TRUE);

recordTerminator();
recordTerminatorWithNewline();

                
END_METHOD

METHOD configureBool : BOOL
  VAR_INPUT
    parameter : t_token_type;
    target : REFERENCE TO BOOL;
    required : BOOL;
    particle : POINTER TO t_particle;
  END_VAR
  VAR
    valueToken : t_token_string;
  END_VAR
                  configureBool := matchArgument(parameter,valueToken);

IF (NOT(configureBool)) THEN
	IF (required) THEN
		executeContextFail(THIS,cExecuteReturnMissingArgument,TRUE);		
	END_IF
	
	RETURN;
END_IF

IF (NOT(gTypeHandler.getBoolFromToken(valueToken,target))) THEN
	executeContextFail(THIS,cExecuteReturnParseParameterError,TRUE);
	RETURN;
END_IF

gSystemServices.Executor.reportParameterUpdates(particle);


                
END_METHOD

METHOD appendTokenPair
  VAR_INPUT
    parameter : t_token_type;
    value : STRING;
    quoted : BOOL;
    comma : BOOL;
  END_VAR
  VAR
    stmp : STRING;
  END_VAR
                  IF (strcmp(value,'')) THEN
	RETURN;
END_IF

lWriteStream.appendPair(gTypeHandler.getTokenForEnum(cEnumTypeTokenType,parameter),value,quoted,comma);

                
END_METHOD

METHOD getNextExecuteCommand : BOOL
                  lError := FALSE;
lExecuteReturn := cExecuteReturnOK;

lExecutionQueueCount := 0;
lExecutionQueueIndex := 0;
lRegisterDepth := 0;

IF (NOT(_getNextExecuteCommand())) THEN
	getNextExecuteCommand := FALSE;
	RETURN;
END_IF

getNextExecuteCommand := TRUE;

IF (lCurrentCommand.command=cTokenNone) THEN
	executeContextFail(THIS,cExecuteReturnExecutionQueueNullParticle,TRUE);		
	RETURN;	
END_IF

IF (lCurrentCommand.particle=0) THEN
	executeContextFail(THIS,cExecuteReturnExecutionQueueNullParticle,TRUE);		
	RETURN;
END_IF

IF (lEnableExecutor) THEN
	IF (matchOption(cExecuteOptionExecutor)) THEN	
		IF (NOT(gSystemServices.Executor.putCommand(lCurrentCommand))) THEN
			executeContextFail(THIS,cExecuteReturnExecutionExecutorFailed,TRUE);	
		END_IF
	
		RETURN;
	END_IF
END_IF

IF ((matchOption(cExecuteOptionRecurse)) OR
	(matchOption(cExecuteOptionSubsystems))) THEN
	lCurrentCommand.particle^.recurse(THIS);
ELSE
	registerParticle(lCurrentCommand.particle);	
END_IF

                
END_METHOD

METHOD matchCommand : BOOL
  VAR_INPUT
    contender : REFERENCE TO t_command_definition;
  END_VAR
  VAR
    i : USINT;
    j : USINT;
  END_VAR
                  IF (lCurrentCommand.command<>contender.command) THEN
	matchCommand := FALSE;
	RETURN;
END_IF

FOR i:=1 TO lCurrentCommand.optionCount DO
	FOR j:=1 TO cExecuteOptionListCount DO
		IF (lCurrentCommand.options[i]=contender.options[j]) THEN
			EXIT;
		END_IF
	END_FOR
	
	IF (j>cExecuteOptionListCount) THEN
		executeContextFail(THIS,cExecuteReturnUnknownOption,TRUE);		
	END_IF
END_FOR

IF (lCurrentCommand.argumentCount<contender.pairMinCount) THEN
	executeContextFail(THIS,cExecuteReturnTooFewArguments,TRUE);		
END_IF

IF (lCurrentCommand.argumentCount>contender.pairMaxCount) THEN
	executeContextFail(THIS,cExecuteReturnTooManyArguments,TRUE);		
END_IF

IF ((contender.readwrite) AND (NOT(lReadWrite))) THEN
	executeContextFail(THIS,cExecuteReturnReadOnly,TRUE);
END_IF

matchCommand := TRUE;

                
END_METHOD

METHOD matchOption : BOOL
  VAR_INPUT
    option : t_execute_option;
  END_VAR
  VAR
    i : USINT;
  END_VAR
                  FOR i:=1 TO lCurrentCommand.optionCount DO
	IF (lCurrentCommand.options[i]=option) THEN
		matchOption := TRUE;
		RETURN;
	END_IF
END_FOR

matchOption := FALSE;

                
END_METHOD

METHOD matchArgument : BOOL
  VAR_INPUT
    parameter : t_token_type;
    value : REFERENCE TO t_token_string;
  END_VAR
  VAR
    i : USINT;
  END_VAR
                  FOR i:=1 TO lCurrentCommand.argumentCount DO
	IF ((lCurrentCommand.arguments[i].parameter=parameter) AND
		(NOT(lCurrentCommand.arguments[i].processed))) THEN
		value := lCurrentCommand.arguments[i].value;
		lCurrentCommand.arguments[i].processed := TRUE;
		
		matchArgument := TRUE;	
		RETURN;
	END_IF
END_FOR
	
matchArgument := FALSE;
                
END_METHOD

METHOD _getNextExecuteCommand : BOOL
                  _getNextExecuteCommand := false;
                
END_METHOD

METHOD appendIdentity
  VAR_INPUT
    particle : POINTER TO t_particle;
  END_VAR
                  IF (particle=0) THEN
	RETURN;
END_IF

recordInitiator();	
appendPair('identity',particle^.lIdentity,TRUE,FALSE);
appendPair('type',particle^.TypeToken,TRUE,TRUE);
appendPair('subsystem',gTypeHandler.getTokenForEnum(cEnumTypeSubsystem,particle^.SubSystem),TRUE,TRUE);
recordTerminatorWithNewline();


                
END_METHOD

PROPERTY EnableExecutor : BOOL
GET
                    EnableExecutor := lEnableExecutor;
                  
END_GET
SET
                    lEnableExecutor := EnableExecutor;
                  
END_SET
END_PROPERTY

PROPERTY WriteStream : POINTER TO t_stream
GET
                    WriteStream := ADR(lWriteStream);
                  
END_GET
END_PROPERTY

PROPERTY ReadWrite : BOOL
GET
                    ReadWrite := lReadWrite;
                  
END_GET
SET
  VAR
    i : USINT;
  END_VAR
                    lReadWrite := ReadWrite;

                  
END_SET
END_PROPERTY

PROPERTY Error : BOOL
GET
                    Error := lError;
                  
END_GET
SET
                    lError := Error;
                  
END_SET
END_PROPERTY

PROPERTY Command : REFERENCE TO t_command_request
GET
                    Command ref= lCurrentCommand;
                  
END_GET
END_PROPERTY

PROPERTY ExecuteReturn : t_execute_return
GET
                    ExecuteReturn := lExecuteReturn;
                  
END_GET
SET
                    IF ((lExecuteReturn=cExecuteReturnOK) or
	(ExecuteReturn=cExecuteReturnOK)) THEN
	lExecuteReturn := ExecuteReturn;
END_IF

                  
END_SET
END_PROPERTY

PROPERTY ExecutionComplete : BOOL
GET
                    ExecutionComplete := ((lExecutionQueueIndex>=lExecutionQueueCount) OR
	(lError));
                  
END_GET
END_PROPERTY

PROPERTY PassComplete : BOOL
GET
                    PassComplete := (lPassCount >= lPassLimit);

                  
END_GET
END_PROPERTY

PROPERTY ArgsUnprocessed : BOOL
GET
  VAR
    i : USINT;
  END_VAR
                    FOR i:=1 TO lCurrentCommand.argumentCount DO
	IF (NOT(lCurrentCommand.arguments[i].processed)) THEN
		ArgsUnprocessed := TRUE;
		RETURN;
	END_IF
END_FOR

ArgsUnprocessed := FALSE;
                  
END_GET
END_PROPERTY

PROPERTY ReportError : BOOL
GET
                    ReportError := lReportError;
                  
END_GET
SET
                    lReportError := ReportError;
                  
END_SET
END_PROPERTY

PROPERTY WrappedResponse : BOOL
GET
                    WrappedResponse := lWrappedResponse;
                  
END_GET
SET
                    lWrappedResponse := WrappedResponse;

IF (WrappedResponse) THEN
	lWriteStream.IndentStr := '';
ELSE
	lWriteStream.IndentStr := '    ';	
END_IF
                  
END_SET
END_PROPERTY
END_FUNCTION_BLOCK

{attribute 'enable_dynamic_creation'}
FUNCTION_BLOCK ExecuteContextExecutor EXTENDS ExecuteContext
  VAR
    lSource : REFERENCE TO Executor;
  END_VAR

            
          

METHOD _getNextExecuteCommand : BOOL
                  IF (__ISVALIDREF(lSource)) THEN
	_getNextExecuteCommand := lSource.getNextExecuteCommand(lCurrentCommand);
ELSE
	_getNextExecuteCommand := FALSE;
END_IF

                
END_METHOD

PROPERTY Source : REFERENCE TO Executor
GET
                    Source ref= lSource;
                  
END_GET
SET
                    lSource REF= Source;
                  
END_SET
END_PROPERTY
END_FUNCTION_BLOCK

{attribute 'enable_dynamic_creation'}
FUNCTION_BLOCK ExecuteContextParse EXTENDS ExecuteContext
  VAR
    lSource : REFERENCE TO ParseConnectionHandler;
  END_VAR

            
          

METHOD _getNextExecuteCommand : BOOL
                  IF (__ISVALIDREF(lSource)) THEN
	_getNextExecuteCommand := lSource.getNextExecuteCommand(lCurrentCommand);
ELSE
	_getNextExecuteCommand := FALSE;
END_IF

                
END_METHOD

PROPERTY Source : REFERENCE TO ParseConnectionHandler
GET
                    Source ref= lSource;
                  
END_GET
SET
                    lSource REF= Source;
                  
END_SET
END_PROPERTY
END_FUNCTION_BLOCK

FUNCTION_BLOCK ExecuteSource
  VAR
    lCommand : t_token_type;
    lOptions : t_options_list;
    lPairs : ARRAY[1..4] OF t_argument;
  END_VAR

            
          

METHOD getNextExecuteCommand : BOOL
  VAR_INPUT
    command : REFERENCE TO t_command_request;
  END_VAR
                  






                
END_METHOD
END_FUNCTION_BLOCK

FUNCTION_BLOCK NonOperationalParticleSet EXTENDS Particle
  VAR CONSTANT
    cNopParticleSetMax : USINT := 64;
  END_VAR
  VAR
    lNonOperationalParticleCount : USINT := 0;
    lNonOperationalParticleSet : ARRAY[1..cNopParticleSetMax] OF t_particle_ptr;
  END_VAR

            
          

METHOD getParticle : POINTER TO t_particle
  VAR_INPUT
    name : REFERENCE TO t_token_string;
    id : t_particle_id;
  END_VAR
  VAR
    i : USINT;
    particle : POINTER TO t_particle;
  END_VAR
                  FOR i:=1 TO lNonOperationalParticleCount DO
	IF (id>0) THEN
		particle := lNonOperationalParticleSet[i]^.getParticle(name,id);
		IF (particle<>0) THEN
			getParticle := particle;
			RETURN;
		END_IF
	ELSE
		IF (strcmp(name,lNonOperationalParticleSet[i]^.lName)) THEN
			getParticle := lNonOperationalParticleSet[i];
			RETURN;
		END_IF		
	END_IF
END_FOR

getParticle := SUPER^.getParticle(name,id);

                
END_METHOD

METHOD initialize
  VAR
    i : USINT;
  END_VAR
                  SUPER^.initialize();

FOR i:=1 TO lNonOperationalParticleCount DO
	IF (lNonOperationalParticleSet[i]^.lParticleId=0) THEN
		lNonOperationalParticleSet[i]^.initialize();
	END_IF
END_FOR
                
END_METHOD

METHOD registerNonOperational
  VAR_INPUT
    particle : t_particle_ptr;
  END_VAR
                  IF (particle=0) THEN
	RETURN;
END_IF

IF (lNonOperationalParticleCount>=cNopParticleSetMax) THEN
	gCodeErrorHandler(pMessage:='NonOperationalParticleSet overflow');
	RETURN;
END_IF

lNonOperationalParticleCount := lNonOperationalParticleCount + 1;
lNonOperationalParticleSet[lNonOperationalParticleCount] := particle;
particle^.Parent := THIS;
//particle^.System REF= System;
particle^.SubSystem := SubSystem;

                
END_METHOD

METHOD identify
  VAR
    i : USINT;
  END_VAR
                  SUPER^.identify();

FOR i:=1 TO lNonOperationalParticleCount DO
	lNonOperationalParticleSet[i]^.identify();
END_FOR

                
END_METHOD

METHOD loadExecutionContext
  VAR_INPUT
    executeContext : POINTER TO ExecuteContext;
  END_VAR
  VAR
    i : USINT;
  END_VAR
                  SUPER^.loadExecutionContext(executeContext);

IF (executeContext=0) THEN
	RETURN;
END_IF

IF (lProceed) THEN
	executeContext^.registerDepthIncrease();
	FOR i:=1 TO lNonOperationalParticleCount DO
		lNonOperationalParticleSet[i]^.loadExecutionContext(executeContext);
	END_FOR
	executeContext^.registerDepthDecrease();
END_IF

                
END_METHOD

METHOD recurse
  VAR_INPUT
    executeContext : POINTER TO ExecuteContext;
  END_VAR
  VAR
    i : USINT;
  END_VAR
                  SUPER^.recurse(executeContext);

IF (NOT(executeContext^.matchOption(cExecuteOptionRecurse))) THEN	
	RETURN;
END_IF

FOR i:=1 TO lNonOperationalParticleCount DO
	lNonOperationalParticleSet[i]^.recurse(executeContext);
END_FOR
                
END_METHOD

METHOD describe
  VAR_INPUT
    executeContext : POINTER TO ExecuteContext;
  END_VAR
  VAR
    i : USINT;
  END_VAR
                  SUPER^.describe(executeContext);

IF (executeContext^.matchOption(cExecuteOptionSyntax)) THEN
	RETURN;
END_IF

IF (executeContext^.matchOption(cExecuteOptionParameter)) THEN
	RETURN;
END_IF

IF (NOT(executeContext^.matchOption(cExecuteOptionChildren))) THEN
	RETURN;
END_IF

executeContext^.append(', ');
executeContext^.WriteStream^.increaseIndent();
executeContext^.formatWithNewlineIndent();
executeContext^.append('"nop-children": [');
executeContext^.WriteStream^.increaseIndent();

FOR i:=1 TO lNonOperationalParticleCount DO
	executeContext^.recordInitiatorWithNewlineIndent();
	executeContext^.appendPair('identity',lNonOperationalParticleSet[i]^.lIdentity,TRUE,FALSE);
	executeContext^.appendPair('type',lNonOperationalParticleSet[i]^.TypeToken,TRUE,TRUE);
	executeContext^.appendPair('subsystem',gTypeHandler.getTokenForEnum(cEnumTypeSubsystem,lNonOperationalParticleSet[i]^.SubSystem),TRUE,TRUE);
	executeContext^.recordTerminator();
	
	IF (i<lNonOperationalParticleCount) THEN
		executeContext^.append(', ');		
	END_IF
END_FOR

executeContext^.WriteStream^.decreaseIndent();
executeContext^.append(']');
executeContext^.WriteStream^.decreaseIndent();

                
END_METHOD

PROPERTY NopSelf : POINTER TO NonOperationalParticleSet
GET
                    NopSelf := THIS;
                  
END_GET
END_PROPERTY

PROPERTY SubSystem : t_subsystem
SET
  VAR
    i : USINT;
  END_VAR
                    IF (lSubSystem=cSubsystemNone) THEN
	lSubSystem := SubSystem;
	
	FOR i:=1 TO lNonOperationalParticleCount DO
		lNonOperationalParticleSet[i]^.SubSystem := lSubSystem;
	END_FOR
END_IF

                  
END_SET
END_PROPERTY

PROPERTY FailSafeMode : BOOL
SET
  VAR
    i : USINT;
  END_VAR
                    SUPER^.FailSafeMode := FailSafeMode;

IF (lProceed) THEN
	FOR i:=1 TO lNonOperationalParticleCount DO
		lNonOperationalParticleSet[i]^.FailSafeMode := FailSafeMode;
	END_FOR		
END_IF

                  
END_SET
END_PROPERTY
END_FUNCTION_BLOCK

FUNCTION_BLOCK OperationalParticleSet EXTENDS NonOperationalParticleSet
  VAR CONSTANT
    cOpParticleSetMax : USINT := 64;
  END_VAR
  VAR
    lOperationalParticleCount : USINT := 0;
    lOperationalParticleSet : ARRAY[1..cOpParticleSetMax] OF t_particle_ptr;
  END_VAR

            
          

METHOD getParticle : POINTER TO t_particle
  VAR_INPUT
    name : REFERENCE TO t_token_string;
    id : t_particle_id;
  END_VAR
  VAR
    i : USINT;
    particle : POINTER TO t_particle;
  END_VAR
                  FOR i:=1 TO lOperationalParticleCount DO
	IF (id>0) THEN
		particle := lOperationalParticleSet[i]^.getParticle(name,id);
		IF (particle<>0) THEN
			getParticle := particle;
			RETURN;
		END_IF
	ELSE
		IF (strcmp(name,lOperationalParticleSet[i]^.lName)) THEN
			getParticle := lOperationalParticleSet[i];
			RETURN;
		END_IF		
	END_IF
END_FOR

getParticle := SUPER^.getParticle(name,id);

                
END_METHOD

METHOD initialize
  VAR
    i : USINT;
  END_VAR
                  SUPER^.initialize();

FOR i:=1 TO lOperationalParticleCount DO
	IF (lOperationalParticleSet[i]^.lParticleId=0) THEN
		lOperationalParticleSet[i]^.initialize();
	END_IF
END_FOR

                
END_METHOD

METHOD operator
  VAR
    i : USINT;
  END_VAR
                  IF (NOT(lProceed)) THEN
	RETURN;
END_IF

FOR i:=1 TO lOperationalParticleCount DO
	IF (lOperationalParticleSet[i]^.lProceed) THEN
		lOperationalParticleSet[i]^.operator();
	END_IF
END_FOR

SUPER^.operator();
                
END_METHOD

METHOD registerOperational
  VAR_INPUT
    particle : t_particle_ptr;
  END_VAR
                  IF (particle=0) THEN
	RETURN;
END_IF

IF (lOperationalParticleCount>=cOpParticleSetMax) THEN
	gCodeErrorHandler(pMessage:='OperationalParticleSet overflow');
	RETURN;
END_IF

lOperationalParticleCount := lOperationalParticleCount + 1;
lOperationalParticleSet[lOperationalParticleCount] := particle;
particle^.Parent := THIS;
//particle^.System REF= System;
particle^.SubSystem := SubSystem;

                
END_METHOD

METHOD identify
  VAR
    i : USINT;
  END_VAR
                  SUPER^.identify();

FOR i:=1 TO lOperationalParticleCount DO
	lOperationalParticleSet[i]^.identify();
END_FOR

                
END_METHOD

METHOD loadExecutionContext
  VAR_INPUT
    executeContext : POINTER TO ExecuteContext;
  END_VAR
  VAR
    i : USINT;
  END_VAR
                  SUPER^.loadExecutionContext(executeContext);

IF (executeContext=0) THEN
	RETURN;
END_IF

IF (lProceed) THEN
	executeContext^.registerDepthIncrease();
	FOR i:=1 TO lOperationalParticleCount DO
		lOperationalParticleSet[i]^.loadExecutionContext(executeContext);
	END_FOR
	executeContext^.registerDepthDecrease();
END_IF

                
END_METHOD

METHOD recurse
  VAR_INPUT
    executeContext : POINTER TO ExecuteContext;
  END_VAR
  VAR
    i : USINT;
  END_VAR
                  SUPER^.recurse(executeContext);

IF (NOT(executeContext^.matchOption(cExecuteOptionRecurse))) THEN	
	RETURN;
END_IF

FOR i:=1 TO lOperationalParticleCount DO
	lOperationalParticleSet[i]^.recurse(executeContext);
END_FOR
                
END_METHOD

METHOD describe
  VAR_INPUT
    executeContext : POINTER TO ExecuteContext;
  END_VAR
  VAR
    i : USINT;
  END_VAR
                  SUPER^.describe(executeContext);

IF (executeContext^.matchOption(cExecuteOptionSyntax)) THEN
	RETURN;
END_IF

IF (executeContext^.matchOption(cExecuteOptionParameter)) THEN
	RETURN;
END_IF

IF (NOT(executeContext^.matchOption(cExecuteOptionChildren))) THEN
	RETURN;
END_IF

executeContext^.append(', ');
executeContext^.WriteStream^.increaseIndent();
executeContext^.formatWithNewlineIndent();
executeContext^.append('"op-children": [');
executeContext^.WriteStream^.increaseIndent();

FOR i:=1 TO lOperationalParticleCount DO
	executeContext^.recordInitiatorWithNewlineIndent();
	executeContext^.appendPair('identity',lOperationalParticleSet[i]^.lIdentity,TRUE,FALSE);
	executeContext^.appendPair('type',lOperationalParticleSet[i]^.TypeToken,TRUE,TRUE);
	executeContext^.appendPair('subsystem',gTypeHandler.getTokenForEnum(cEnumTypeSubsystem,lOperationalParticleSet[i]^.SubSystem),TRUE,TRUE);
	executeContext^.recordTerminator();
	
	IF (i<lOperationalParticleCount) THEN
		executeContext^.append(', ');		
	END_IF
END_FOR

executeContext^.WriteStream^.decreaseIndent();
executeContext^.append(']');
executeContext^.WriteStream^.decreaseIndent();


                
END_METHOD

PROPERTY OpSelf : POINTER TO OperationalParticleSet
GET
                    OpSelf := THIS;
                  
END_GET
END_PROPERTY

PROPERTY ChildrenOK : BOOL
GET
  VAR
    i : USINT;
  END_VAR
                    ChildrenOK := TRUE;

FOR i:=1 TO lOperationalParticleCount DO
	IF (NOT(lOperationalParticleSet[i]^.OK)) THEN
		ChildrenOK := FALSE;
	END_IF
END_FOR

                  
END_GET
END_PROPERTY

PROPERTY SubSystem : t_subsystem
SET
  VAR
    i : USINT;
  END_VAR
                    IF (lSubSystem=cSubsystemNone) THEN
	lSubSystem := SubSystem;
	
	FOR i:=1 TO lOperationalParticleCount DO
		lOperationalParticleSet[i]^.SubSystem := lSubSystem;
	END_FOR

	FOR i:=1 TO lNonOperationalParticleCount DO
		lNonOperationalParticleSet[i]^.SubSystem := lSubSystem;
	END_FOR
END_IF

                  
END_SET
END_PROPERTY

PROPERTY FailSafeMode : BOOL
SET
  VAR
    i : USINT;
  END_VAR
                    SUPER^.FailSafeMode := FailSafeMode;

IF (lProceed) THEN
	FOR i:=1 TO lOperationalParticleCount DO
		lOperationalParticleSet[i]^.FailSafeMode := FailSafeMode;
	END_FOR
END_IF

                  
END_SET
END_PROPERTY
END_FUNCTION_BLOCK

FUNCTION_BLOCK Particle
  VAR_INPUT
    lProceed : BOOL := TRUE;
    lFailSafeConfig : BOOL := FALSE;
    lParticleId : t_particle_id := 0;
    lIdentity : t_long_string;
    lFeature : BOOL := TRUE;
  END_VAR
  VAR
    lFBCount : USINT := 0;
    lParent : POINTER TO t_particle := 0;
    lName : t_name := sDefaultName;
    lDescription : t_long_string;
    lSubSystem : t_subsystem := cSubsystemNone;
    lCnt : USINT := 0;
  END_VAR

            
          

METHOD configure
  VAR_INPUT
    executeContext : POINTER TO ExecuteContext;
  END_VAR
                  IF (executeContext^.configureBool(cTokenProceed,lProceed,FALSE,THIS)) THEN
	RETURN;
END_IF

IF (executeContext^.configureBool(cTokenFailSafeConfig,lFailSafeConfig,FALSE,THIS)) THEN
	RETURN;
END_IF

executeContextFail(executeContext,cExecuteReturnUnknownParameter,TRUE);

                
END_METHOD

METHOD describe
  VAR_INPUT
    executeContext : POINTER TO ExecuteContext;
  END_VAR
                  gParticleDebugIdB := lParticleId;

IF (executeContext^.matchOption(cExecuteOptionSyntax)) THEN
	executeContext^.describeSyntaxExecutable(sCommandDescribe);
	executeContext^.describeSyntaxExecutable(sCommandVerify);
	executeContext^.describeSyntaxExecutable(sCommandIdentify);
	executeContext^.describeSyntaxExecutable(sCommandSetFailSafeMode);
	executeContext^.describeSyntaxExecutable(sCommandClearFailSafeMode);

	executeContext^.describeSyntaxConfigurable(cValueStyleParameter,cTokenProceed,cDataTypeBool,cEnumTypeNone,'',cDescriptionProceed);
	executeContext^.describeSyntaxConfigurable(cValueStyleParameter,cTokenFailSafeConfig,cDataTypeBool,cEnumTypeNone,'',cDescriptionFailSafeConfig);

	RETURN;
END_IF

IF (executeContext^.matchOption(cExecuteOptionParameter)) THEN
	executeContext^.describeParameter(cValueStyleConfigurable,lIdentity,cTokenProceed,gTypeHandler.getTokenForBool(lProceed),cDataTypeBool,cEnumTypeNone,'',cDescriptionProceed);
	executeContext^.describeParameter(cValueStyleConfigurable,lIdentity,cTokenFailSafeConfig,gTypeHandler.getTokenForBool(lFailSafeConfig),cDataTypeBool,cEnumTypeNone,'',cDescriptionFailSafeConfig);
	
	RETURN;
END_IF

executeContext^.appendPair('identity',lIdentity,TRUE,FALSE);
executeContext^.appendPair('type',TypeToken,TRUE,TRUE);
executeContext^.appendPair('subsystem',gTypeHandler.getTokenForEnum(cEnumTypeSubsystem,SubSystem),TRUE,TRUE);
executeContext^.appendPair('description',lDescription,TRUE,TRUE);

IF (executeContext^.matchOption(cExecuteOptionVerbose)) THEN
	executeContext^.appendTokenPair(cTokenProceed,gTypeHandler.getTokenForBool(lProceed),FALSE,TRUE);
	executeContext^.appendTokenPair(cTokenFailSafeConfig,gTypeHandler.getTokenForBool(lFailSafeConfig),FALSE,TRUE);
END_IF


                
END_METHOD

METHOD execute
  VAR_INPUT
    executeContext : POINTER TO ExecuteContext;
  END_VAR
  VAR
    token : t_token_string;
  END_VAR
                  IF (executeContext=0) THEN
	RETURN;
END_IF

IF (executeContext^.matchCommand(sCommandConfigure)) THEN
	configure(executeContext);
	RETURN;
END_IF

IF (executeContext^.matchCommand(sCommandVerify)) THEN
	verify(executeContext);
	RETURN;
END_IF

IF (executeContext^.matchCommand(sCommandSetFailSafeMode)) THEN
	FailSafeMode := TRUE;
	RETURN;
END_IF

IF (executeContext^.matchCommand(sCommandClearFailSafeMode)) THEN
	FailSafeMode := FALSE;
	RETURN;
END_IF

IF (executeContext^.matchCommand(sCommandDescribe)) THEN

	IF (executeContext^.matchOption(cExecuteOptionSyntax)) THEN
		executeContext^.recordInitiator();
		executeContext^.appendPair('identity',lIdentity,TRUE,FALSE);
		executeContext^.append(',"syntax": [');
		describe(executeContext);
		executeContext^.append(']');
		executeContext^.recordTerminatorWithNewline();

		RETURN;
	END_IF
	
	IF (executeContext^.matchOption(cExecuteOptionParameter)) THEN
		describe(executeContext);
		RETURN;
	END_IF
		
	executeContext^.recordInitiator();
	describe(executeContext);
	executeContext^.recordTerminatorWithNewline();

	RETURN;
END_IF

IF (executeContext^.matchCommand(sCommandIdentify)) THEN
	executeContext^.appendIdentity(THIS);
	RETURN;
END_IF

executeContextFail(executeContext,cExecuteReturnUnknownCommand,TRUE);

                
END_METHOD

METHOD getParticle : POINTER TO t_particle
  VAR_INPUT
    name : REFERENCE TO t_token_string;
    id : t_particle_id;
  END_VAR
                  getParticle := 0;

IF (id>0) THEN
	IF (id=lParticleId) THEN
		getParticle := THIS;
	END_IF
	
	RETURN;
END_IF

IF (strcmp(name,lName)) THEN
	getParticle := THIS;
	RETURN;
END_IF

IF (strcmp(name,'this')) THEN
	getParticle := THIS;
	RETURN;
END_IF



                
END_METHOD

METHOD identify
                  IF (lParent<>0) THEN
	IF ((find(lIdentity,'/')>0) OR
		(lParent^.lFeature)) THEN
		lIdentity := CONCAT(lParent^.lIdentity,'/');
	ELSE
		lIdentity := CONCAT(lParent^.lIdentity,'.');
	END_IF
	lIdentity := CONCAT(lIdentity,lName);

	RETURN;
END_IF

lIdentity := CONCAT(gNameSpace,'.');
lIdentity := CONCAT(lIdentity,lName);

                
END_METHOD

METHOD initialize
                  IF (lParticleId<>0) THEN
	RETURN;
END_IF

Name := TypeToken;

sLastParticleId := sLastParticleId + 1;
lParticleId := sLastParticleId;

                
END_METHOD

METHOD operator
                  lCnt := lCnt + 1;

                
END_METHOD

METHOD verify
  VAR_INPUT
    executeContext : POINTER TO ExecuteContext;
  END_VAR
                  IF (lParticleId=0) THEN
	executeContext^.describeVerify(lIdentity,FALSE,'zero ParticleId');
END_IF

IF (strcmp(lName,sDefaultName)) THEN
	executeContext^.describeVerify(lIdentity,FALSE,'default name');
END_IF

IF (strcmp(sParticle,TypeToken)) THEN
	executeContext^.describeVerify(lIdentity,FALSE,'default type');
END_IF

IF (SubSystem=cSubsystemNone) THEN
	executeContext^.describeVerify(lIdentity,FALSE,'default subsystem');
END_IF

//IF (NOT(__ISVALIDREF(_System)))THEN
//	executeContext^.describeVerify(lIdentity,FALSE,'null System reference');
//END_IF
                
END_METHOD

METHOD loadExecutionContext
  VAR_INPUT
    executeContext : POINTER TO ExecuteContext;
  END_VAR
                  IF (executeContext=0) THEN
	RETURN;
END_IF

executeContext^.registerParticle(THIS);

                
END_METHOD

METHOD recurse
  VAR_INPUT
    executeContext : POINTER TO ExecuteContext;
  END_VAR
                  IF (executeContext=0) THEN
	RETURN;
END_IF

executeContext^.registerParticle(THIS);	

                
END_METHOD

METHOD FB_Init : BOOL
  VAR_INPUT
    bInitRetains : BOOL;
    bInCopyCode : BOOL;
  END_VAR
                  lFBCount := lFBCount + 1;
// {attribute 'enable-dynamic-creation'}

//allocateLongString(lIdentity);
lIdentity REF= _defaultLongString;

                
END_METHOD

PROPERTY Name : t_name
GET
                    Name := lName;
                  
END_GET
SET
                    IF ((find(Name,'.')>0) OR
	(find(Name,'/')>0)) THEN
	gCodeErrorHandler(pMessage:='Illegal . or / character in name');
	RETURN;
END_IF

IF (strcmp(lName,sDefaultName)) THEN
	lName := Name;
	identify();
END_IF

                  
END_SET
END_PROPERTY

PROPERTY OK : BOOL
GET
  VAR
    i : USINT;
  END_VAR
                    OK := TRUE;

                  
END_GET
END_PROPERTY

PROPERTY Parent : POINTER TO t_particle
GET
                    Parent := lParent;
                  
END_GET
SET
                    lParent := Parent;
identify();

                  
END_SET
END_PROPERTY

PROPERTY SubSystem : t_subsystem
GET
                    SubSystem := lSubSystem;
                  
END_GET
SET
                    IF (lSubSystem=cSubsystemNone) THEN
	lSubSystem := SubSystem;
END_IF

                  
END_SET
END_PROPERTY

PROPERTY TypeToken : t_medium_string
GET
                    TypeToken := sParticle;

                  
END_GET
END_PROPERTY

PROPERTY FailSafeMode : BOOL
SET
                    IF (FailSafeMode) THEN
	lProceed := lFailSafeConfig;

	gSystemServices.PLC.setFailSafeMode();
ELSE
	lProceed := TRUE;
END_IF

                  
END_SET
END_PROPERTY
END_FUNCTION_BLOCK

FUNCTION_BLOCK PersistentCommand EXTENDS PersistentValue
  VAR
    lValue : t_command_store;
  END_VAR

            
          

METHOD initialize
                  lData := ADR(lValue);
lCount := SIZEOF(lValue);

SUPER^.initialize();

                
END_METHOD

PROPERTY Value : t_command_store
GET
                    Value := lValue;

                  
END_GET
SET
  VAR
    i : USINT;
    equal : BOOL := TRUE;
  END_VAR
                    IF ((Value.argumentCount=lValue.argumentCount) AND
	(Value.command=lValue.command) AND
	(Value.optionCount=lValue.optionCount) AND
	(Value.particle=lValue.particle)) THEN
	
	FOR i:=1 TO lValue.argumentCount DO
		IF (NOT((Value.arguments[i].parameter=lValue.arguments[i].parameter) AND
			(Value.arguments[i].value=lValue.arguments[i].value))) THEN
			equal := FALSE;		
		END_IF
	END_FOR
	
	FOR i:=1 TO lValue.optionCount DO
		IF (NOT(Value.options[i]=lValue.options[i])) THEN
			equal := FALSE;		
		END_IF
	END_FOR

	IF (equal) THEN
		RETURN;
	END_IF
END_IF

FOR i:=Value.optionCount TO cExecuteOptionListCount DO
	Value.options[i] := 0;
END_FOR

FOR i:=Value.argumentCount TO cExecuteArgumentListCount DO
	Value.arguments[i].parameter := 0;
	Value.arguments[i].value := '';
	Value.arguments[i].processed := FALSE;
END_FOR

lValue := Value;
write();
                  
END_SET
END_PROPERTY

PROPERTY Valid : BOOL
GET
                    Valid := (lValue.particle<>0);
                  
END_GET
END_PROPERTY
END_FUNCTION_BLOCK

FUNCTION executeContextFail
  VAR_INPUT
    executeContext : POINTER TO ExecuteContext;
    reason : t_execute_return;
    abort : BOOL;
  END_VAR

            IF (executeContext=0) THEN
	RETURN;
END_IF

executeContext^.ExecuteReturn := reason;

IF (abort) THEN
	executeContext^.Error := TRUE;
END_IF

          
END_FUNCTION

FUNCTION notificationSkippingConfiguration
  VAR_INPUT
    particle : POINTER TO Particle;
    parameter : REFERENCE TO t_token_string;
    value : REFERENCE TO t_token_string;
    writeStream : POINTER TO t_stream;
  END_VAR

            IF (writeStream=0) THEN
	RETURN;
END_IF

writeStream^.append(particle^.lIdentity);
writeStream^.append(' skipping <');	
writeStream^.append(parameter);	
writeStream^.append('>=<');	
writeStream^.append(value);	
writeStream^.append('>');
writeStream^.newline();
          
END_FUNCTION

FUNCTION_BLOCK ReportableChannel EXTENDS OperationalParticleSet
  VAR
    lReportableChannelManager : POINTER TO ReportableChannelManager := 0;
    lEnabled : BOOL := FALSE;
    lCount : ULINT := 0;
    lCountPrevious : ULINT := 0;
    lRate : UINT := 0;
    lChannelMask : t_channel_mask;
    lReportEvent : BOOL := TRUE;  (* lEventCount: ULINT:= 0; lActiveRisingCount: ULINT:= 0; lUnsuppressRisingCount: ULINT:= 0; lUnsuppressFallingCount: ULINT:= 0; lStateExpiredCount: ULINT:= 0; *)
    lReportEventWhenSuppressed : BOOL := FALSE;
    lReportActiveRising : BOOL := TRUE;
    lReportActiveRisingWhenSuppressed : BOOL := FALSE;
    lReportUnsuppressRising : BOOL := TRUE;
    lReportUnsuppressFalling : BOOL := TRUE;
    lReportEach : BOOL := FALSE;
    lReportEachWhenSuppressed : BOOL := FALSE;
    lReportStateExpired : BOOL := TRUE;
    lReportStateExpiredWhenSuppressed : BOOL := FALSE;
  END_VAR

            
          

METHOD _reportEvent
  VAR_INPUT
    event : POINTER TO t_reportableevent;
  END_VAR
                  ;

                
END_METHOD

METHOD _reportState
  VAR_INPUT
    state : POINTER TO t_reportablestate;
    expired : BOOL;
  END_VAR
                  ;

                
END_METHOD

METHOD _reportStateExpired
  VAR_INPUT
    state : POINTER TO t_reportablestate;
  END_VAR
                  ;

                
END_METHOD

METHOD initialize
                  IF (lReportableChannelManager=0) THEN
	gCodeErrorHandler(pMessage:=CONCAT('null pointer in ',lIdentity));
END_IF

SUPER^.initialize();

lCount := 0;

                
END_METHOD

METHOD initializeChannel
  VAR_INPUT
    reportableChannelManager : POINTER TO ReportableChannelManager;
  END_VAR
                  lReportableChannelManager := reportableChannelManager;

                
END_METHOD

METHOD operator
                  IF (gSystemServices.Cycle.IntegralClockTick) THEN
	lRate := ULINT_TO_UINT(lCount - lCountPrevious);
	lCountPrevious := lCount;
END_IF

SUPER^.operator();
                
END_METHOD

METHOD reportEvent
  VAR_INPUT
    event : POINTER TO t_reportableevent;
  END_VAR
                  IF (event^.Override) THEN
	RETURN;
END_IF

IF (NOT(lEnabled)) THEN
	RETURN;
END_IF

IF (NOT(fCheckChannelMask(event^.ChannelMask,lChannelMask))) THEN
	RETURN;
END_IF

IF ((lReportEvent) AND
	((NOT(event^.ResolvedSuppress)) OR
	(lReportEventWhenSuppressed))) THEN
	//lEventCount := lEventCount + 1;
	lCount := lCount + 1;
	_reportEvent(event);

	RETURN;
END_IF


                
END_METHOD

METHOD reportState
  VAR_INPUT
    state : POINTER TO t_reportablestate;
  END_VAR
                  IF (state^.Override) THEN
	RETURN;
END_IF

IF (NOT(lEnabled)) THEN
	RETURN;
END_IF

IF (NOT(fCheckChannelMask(state^.ChannelMask,lChannelMask))) THEN
	RETURN;
END_IF

IF ((state^.ActiveRising) AND
	(lReportActiveRising) AND
	((NOT(state^.ResolvedSuppress)) OR
	(lReportActiveRisingWhenSuppressed))) THEN
	//lActiveRisingCount := lActiveRisingCount + 1;
	lCount := lCount + 1;
	_reportState(state,FALSE);

	RETURN;
END_IF

IF ((state^.UnsuppressRising) AND
	(lReportUnsuppressRising)) THEN
	//lUnsuppressRisingCount := lUnsuppressRisingCount + 1;
	lCount := lCount + 1;
	//_reportStateUnsuppressRising(state);
	_reportState(state,FALSE);

	RETURN;
END_IF

(*IF ((state^.UnsuppressFalling) AND
	(lReportUnsuppressFalling)) THEN
	lUnsuppressFallingCount := lUnsuppressFallingCount + 1;
	lCount := lCount + 1;
	_reportStateUnsuppressFalling(state);

	RETURN;
END_IF

IF ((lReportEach) AND
	((NOT(state^.ResolvedSuppress)) OR
	(lReportEachWhenSuppressed))) THEN
	lCount := lCount + 1;
	_reportState(state);

	RETURN;	
END_IF*)

                
END_METHOD

METHOD reportStateExpired
  VAR_INPUT
    state : POINTER TO t_reportablestate;
  END_VAR
                  IF (state^.Override) THEN
	RETURN;
END_IF

IF (NOT(lEnabled)) THEN
	RETURN;
END_IF

IF (NOT(fCheckChannelMask(state^.ChannelMask,lChannelMask))) THEN
	RETURN;
END_IF

IF ((lReportStateExpired) AND
	((NOT(state^.ResolvedSuppress)) OR
	(lReportStateExpiredWhenSuppressed))) THEN
	//lStateExpiredCount := lStateExpiredCount + 1;
	lCount := lCount + 1;
	_reportState(state,true);

	RETURN;
END_IF

                
END_METHOD

METHOD _reportStateActiveRising
  VAR_INPUT
    state : POINTER TO t_reportablestate;
  END_VAR
                  ;

                
END_METHOD

METHOD _reportStateUnsuppressRising
  VAR_INPUT
    state : POINTER TO t_reportablestate;
  END_VAR
                  ;

                
END_METHOD

METHOD _reportStateUnsuppressFalling
  VAR_INPUT
    state : POINTER TO t_reportablestate;
  END_VAR
                  ;

                
END_METHOD

PROPERTY ChannelMask : t_channel_mask
GET
                    ChannelMask := lChannelMask;
                  
END_GET
SET
                    lChannelMask := ChannelMask;
                  
END_SET
END_PROPERTY

PROPERTY Count : ULINT
GET
                    Count := lCount;
                  
END_GET
END_PROPERTY

PROPERTY Enabled : BOOL
GET
                    Enabled := lEnabled;

                  
END_GET
SET
                    lEnabled := Enabled;
                  
END_SET
END_PROPERTY

PROPERTY Rate : UINT
GET
                    Rate := lRate;
                  
END_GET
END_PROPERTY

PROPERTY ChannelConnected : BOOL
GET
                    ChannelConnected := false;
                  
END_GET
END_PROPERTY

PROPERTY TypeToken : t_medium_string
GET
                    TypeToken := 'RepChannel';
                  
END_GET
END_PROPERTY
END_FUNCTION_BLOCK

FUNCTION_BLOCK ReportableChannelManager EXTENDS OperationalParticleSet
  VAR_INPUT
    lReportableStateManager : ReportableStateManager;
  END_VAR
  VAR
    lChannels : t_channel_set;
    lChannelCount : USINT := 0;
    lChannelMaskDefaultEvent : UINT := 0;
    lChannelMaskDefaultState : UINT := 0;
    lChannelMaskDefaultParticleReporterEvent : UINT := 0;
    lChannelMaskDefaultRoutedEvent : UINT := 0;
    lChannelMaskDefaultRoutedState : UINT := 0;
  END_VAR

            
          

METHOD initialize
                  

registerOperational(ADR(lReportableStateManager));
lReportableStateManager.initializeStateManager(THIS);

SUPER^.initialize();
SubSystem := cSubsystemMachine;

                
END_METHOD

METHOD registerChannel
  VAR_INPUT
    channel : POINTER TO t_channel;
  END_VAR
                  IF (channel=0) THEN
	RETURN;
END_IF

IF (lChannelCount>8) THEN
	gCodeErrorHandler(pMessage:='Reportable channel register overflow');
	RETURN;
END_IF

lChannelCount := lChannelCount + 1;
lChannels[lChannelCount] := channel;

// assume will not fail
registerOperational(channel);

channel^.initializeChannel(THIS);
                
END_METHOD

METHOD report
  VAR_INPUT
    reportable : POINTER TO t_reportable;
  END_VAR
                  IF (reportable=0) THEN
	RETURN;
END_IF

reportable^._report();

                
END_METHOD

METHOD reportEvent
  VAR_INPUT
    event : POINTER TO t_reportableevent;
  END_VAR
  VAR
    i : USINT;
  END_VAR
                  report(event);

(*IF (event^.ResolvedSuppress) THEN
	RETURN;
END_IF*)

FOR i:=1 TO lChannelCount DO
	lChannels[i]^.reportEvent(event);
END_FOR

                
END_METHOD

METHOD reportState
  VAR_INPUT
    state : POINTER TO t_reportablestate;
  END_VAR
  VAR
    i : USINT;
  END_VAR
                  IF (state=0) THEN
	RETURN;
END_IF

state^.raise();
report(state);
lReportableStateManager.raise(state);

(*IF ((state^.ResolvedSuppress) AND
	(NOT(state^.UnsuppressFalling))) THEN
	RETURN;
END_IF*)

FOR i:=1 TO lChannelCount DO
	lChannels[i]^.reportState(state);
END_FOR

                
END_METHOD

METHOD reportStateContextChanged
  VAR_INPUT
    state : POINTER TO t_reportablestate;
  END_VAR
  VAR
    i : USINT;
  END_VAR
                  IF (state=0) THEN
	RETURN;
END_IF

(*IF (state^.ResolvedSuppress) THEN
	RETURN;
END_IF*)

FOR i:=1 TO lChannelCount DO
	lChannels[i]^.reportState(state);
END_FOR
                
END_METHOD

METHOD reportStateExpired
  VAR_INPUT
    state : POINTER TO t_reportablestate;
  END_VAR
  VAR
    i : USINT;
  END_VAR
                  state^.clear();

(*IF (state^.ResolvedSuppress) THEN
	RETURN;
END_IF*)

FOR i:=1 TO lChannelCount DO
	lChannels[i]^.reportStateExpired(state);
END_FOR

                
END_METHOD

METHOD routeEvent
  VAR_INPUT
    event : POINTER TO t_reportableevent;
  END_VAR
  VAR
    i : USINT;
  END_VAR
                  (*IF (event^.ResolvedSuppress) THEN
	RETURN;
END_IF*)

FOR i:=1 TO lChannelCount DO
	lChannels[i]^.reportEvent(event);
END_FOR

                
END_METHOD

METHOD routeState
  VAR_INPUT
    state : POINTER TO t_reportablestate;
  END_VAR
  VAR
    i : USINT;
  END_VAR
                  (*IF (state^.ResolvedSuppress) THEN
	RETURN;
END_IF*)

FOR i:=1 TO lChannelCount DO
	lChannels[i]^.reportState(state);
END_FOR

                
END_METHOD

METHOD routeStateExpired
  VAR_INPUT
    state : POINTER TO t_reportablestate;
  END_VAR
  VAR
    i : USINT;
  END_VAR
                  (*IF (state^.ResolvedSuppress) THEN
	RETURN;
END_IF*)

FOR i:=1 TO lChannelCount DO
	lChannels[i]^.reportStateExpired(state);
END_FOR

                
END_METHOD

METHOD configure
  VAR_INPUT
    executeContext : POINTER TO ExecuteContext;
  END_VAR
  VAR
    b : BOOL;
  END_VAR
                  IF (gSystemServices.Initialized) THEN
	IF (executeContext^.configureBool(cTokenFailSafeConfig,b,FALSE,0)) THEN
		RETURN;
	END_IF
END_IF

SUPER^.configure(executeContext);



                
END_METHOD

PROPERTY ChannelMaskDefaultEvent : UINT
GET
                    ChannelMaskDefaultEvent := lChannelMaskDefaultEvent;

                  
END_GET
SET
                    lChannelMaskDefaultEvent := ChannelMaskDefaultEvent;

                  
END_SET
END_PROPERTY

PROPERTY ChannelMaskDefaultState : UINT
GET
                    ChannelMaskDefaultState := lChannelMaskDefaultState;
                  
END_GET
SET
                    lChannelMaskDefaultState := ChannelMaskDefaultState;
                  
END_SET
END_PROPERTY

PROPERTY TypeToken : t_medium_string
GET
                    TypeToken := 'Reporting';
                  
END_GET
END_PROPERTY

PROPERTY ChannelMaskDefaultRoutedState : UINT
GET
                    ChannelMaskDefaultRoutedState := lChannelMaskDefaultRoutedState;

                  
END_GET
SET
                    lChannelMaskDefaultRoutedState := ChannelMaskDefaultRoutedState;

                  
END_SET
END_PROPERTY

PROPERTY ChannelMaskDefaultRoutedEvent : UINT
GET
                    ChannelMaskDefaultRoutedEvent := lChannelMaskDefaultRoutedEvent;

                  
END_GET
SET
                    lChannelMaskDefaultRoutedEvent := ChannelMaskDefaultRoutedEvent;

                  
END_SET
END_PROPERTY

PROPERTY ChannelConnected : BOOL
GET
  VAR
    i : USINT;
  END_VAR
                    FOR i:=1 TO lChannelCount DO
	IF (lChannels[i]^.ChannelConnected) THEN
		ChannelConnected := TRUE;
		RETURN;
	END_IF
END_FOR

ChannelConnected := FALSE;
                  
END_GET
END_PROPERTY

PROPERTY ChannelMaskDefaultParticleReporterEvent : UINT
GET
                    ChannelMaskDefaultParticleReporterEvent := lChannelMaskDefaultParticleReporterEvent;

                  
END_GET
SET
                    lChannelMaskDefaultParticleReporterEvent := ChannelMaskDefaultParticleReporterEvent;

                  
END_SET
END_PROPERTY
END_FUNCTION_BLOCK

FUNCTION_BLOCK ReportableChannelUIR EXTENDS ReportableChannel
  VAR CONSTANT
    cCQueueMax : UINT := 255;
  END_VAR
  VAR
    lOverflow : BOOL;
    lQueue : ARRAY[1..cCQueueMax] OF t_ui_reportable;
    lQueueCount : UINT := 0;
    lPopIndex : UINT := 1;
    lPushIndex : UINT := 1;
    lLatestCycle : t_ui_reportable;
    lForcePush : BOOL := FALSE;
    lPopCount : UINT := 0;
    lPushCount : UINT := 0;
    lCycleIndex : UINT := 1;
    a : USINT := 0;
    b : USINT := 0;
    c : USINT := 0;
  END_VAR

            
          

METHOD _reportEvent
  VAR_INPUT
    event : POINTER TO t_reportableevent;
  END_VAR
  VAR
    i : USINT;
  END_VAR
                  push(0,event^.Code,event^.SubSystem,TRUE);

                
END_METHOD

METHOD _reportStateExpired
  VAR_INPUT
    state : POINTER TO t_reportablestate;
  END_VAR
  VAR
    i : USINT;
  END_VAR
                  push(state^.Code,0,state^.SubSystem,FALSE);


                
END_METHOD

METHOD initialize
                  SUPER^.initialize();

lQueueCount := 0;
lPopIndex := 1;
lPushIndex := 1;

                
END_METHOD

METHOD _reportState
  VAR_INPUT
    state : POINTER TO t_reportablestate;
    expired : BOOL;
  END_VAR
                  push(state^.Code,0,state^.SubSystem,TRUE);

                
END_METHOD

METHOD popOrCycle : POINTER TO t_ui_reportable
  VAR
    state : POINTER TO t_reportablestate;
  END_VAR
                  a := a+ 1;

lCycleIndex := MAX(lCycleIndex,1);

IF (lQueueCount=0) THEN
	state := lReportableChannelManager^.lReportableStateManager.cycle(lChannelMask,ADR(lCycleIndex),TRUE);
	IF (state=0) THEN
		popOrCycle := 0;
b:= b+ 1;
		RETURN;
	END_IF
	
	_reportState(state,FALSE);
END_IF

c := c+ 1;
popOrCycle := pop();

                
END_METHOD

METHOD push
  VAR_INPUT
    state : t_state_code;
    event : t_event_code;
    subsystem : t_subsystem;
    active : BOOL;
  END_VAR
                  IF (lQueueCount>=cCQueueMax) THEN
	lOverflow := TRUE;
	RETURN;
END_IF

lQueue[lPushIndex].state := state;
lQueue[lPushIndex].event := event;
lQueue[lPushIndex].subsystem := subsystem;
lQueue[lPushIndex].active := active;
lQueue[lPushIndex].valid := TRUE;

lOverflow := FALSE;
lQueueCount := lQueueCount + 1;
lPushCount := lPushCount + 1;

lPushIndex := lPushIndex + 1;
IF (lPushIndex>cCQueueMax) THEN
	lPushIndex := 1;
END_IF
                
END_METHOD

METHOD pop : POINTER TO t_ui_reportable
                  IF (lQueueCount=0) THEN
	pop := 0;
	RETURN;
END_IF

pop := ADR(lQueue[lPopIndex]);
lPopCount := lPopCount + 1;

lQueueCount := lQueueCount - 1;
lPopIndex := lPopIndex + 1;
IF (lPopIndex>cCQueueMax) THEN
	lPopIndex := 1;
END_IF
                
END_METHOD

METHOD _reportStateActiveRising
  VAR_INPUT
    state : POINTER TO t_reportablestate;
  END_VAR
                  _reportState(state,FALSE);

                
END_METHOD

METHOD _reportStateUnsuppressFalling
  VAR_INPUT
    state : POINTER TO t_reportablestate;
  END_VAR
                  _reportStateExpired(state);

                
END_METHOD

METHOD _reportStateUnsuppressRising
  VAR_INPUT
    state : POINTER TO t_reportablestate;
  END_VAR
                  _reportState(state,FALSE);


                
END_METHOD

PROPERTY Overflow : BOOL
GET
                    Overflow := lOverflow;
                  
END_GET
END_PROPERTY

PROPERTY TypeToken : t_medium_string
GET
                    TypeToken := 'RepChanUIR';
                  
END_GET
END_PROPERTY
END_FUNCTION_BLOCK

FUNCTION_BLOCK ReportableEvent EXTENDS Reportable
  VAR
    lCode : t_event_code;
  END_VAR

            
          

METHOD initialize
                  SUPER^.initialize();

lChannelMask := gSystemServices.ReportableChannelManager.ChannelMaskDefaultEvent;


                
END_METHOD

METHOD initializeEvent
  VAR_INPUT
    p : POINTER TO t_particle_nop;
    name : t_token_string;
    code : t_event_code;
  END_VAR
                  lCode := code;

IF (name='') THEN
	Name := getStringForEventCode(Code);
ELSE
	Name := name;
END_IF

IF (p=0) THEN
	gCodeErrorHandler(pMessage:='initializing reportable with null t_particle_nop');
	RETURN;
END_IF

p^.registerNonOperational(THIS);


                
END_METHOD

METHOD report
  VAR_INPUT
    override : BOOL;
  END_VAR
                  IF ((override) OR 
	(Override)) THEN
	RETURN;
END_IF

SUPER^.report(override);

gSystemServices.ReportableChannelManager.reportEvent(NopSelf);

                
END_METHOD

METHOD initializeEventOp
  VAR_INPUT
    p : POINTER TO t_particle_op;
    name : t_token_string;
    code : t_event_code;
  END_VAR
                  lCode := code;

IF (name='') THEN
	Name := getStringForEventCode(Code);
ELSE
	Name := name;
END_IF

IF (p=0) THEN
	gCodeErrorHandler(pMessage:='initializing reportable with null t_particle_op');
	RETURN;
END_IF

p^.registerOperational(THIS);

                
END_METHOD

METHOD execute
  VAR_INPUT
    executeContext : POINTER TO ExecuteContext;
  END_VAR
                  IF (executeContext^.matchCommand(sCommandTrigger)) THEN	
	trigger(FALSE);
	RETURN;
END_IF

SUPER^.execute(executeContext);

                
END_METHOD

METHOD describe
  VAR_INPUT
    executeContext : POINTER TO ExecuteContext;
  END_VAR
                  SUPER^.describe(executeContext);

IF (executeContext^.matchOption(cExecuteOptionSyntax)) THEN
	executeContext^.describeSyntaxExecutable(sCommandTrigger);
	RETURN;
END_IF

IF (executeContext^.matchOption(cExecuteOptionParameter)) THEN	
	RETURN;
END_IF

executeContext^.appendPair('style','event',TRUE,TRUE);

                
END_METHOD

PROPERTY Code : t_event_code
GET
                    Code := lCode;
                  
END_GET
SET
                    lCode := Code;
                  
END_SET
END_PROPERTY

PROPERTY TypeToken : t_medium_string
GET
                    TypeToken := 'Event';
                  
END_GET
END_PROPERTY
END_FUNCTION_BLOCK

FUNCTION_BLOCK PendingBool
  VAR
    lDefault : BOOL := FALSE;
    lValue : BOOL := FALSE;
    lPending : BOOL := FALSE;
  END_VAR

            
          

METHOD operator
  VAR_INPUT
    override : BOOL;
  END_VAR
                  IF (override) THEN
	lValue := lDefault;
ELSE
	lValue := lPending;
END_IF

lPending := lDefault;

                
END_METHOD

PROPERTY Default : BOOL
GET
                    Default := lDefault;
                  
END_GET
SET
                    lDefault := Default;
                  
END_SET
END_PROPERTY

PROPERTY Pending : BOOL
GET
                    Pending := lPending;
                  
END_GET
SET
                    IF (NOT(Pending=lDefault)) THEN
	lPending := Pending;
END_IF



                  
END_SET
END_PROPERTY

PROPERTY Value : BOOL
GET
                    Value := lValue;
                  
END_GET
END_PROPERTY
END_FUNCTION_BLOCK

FUNCTION_BLOCK PendingChargeQualifier
  VAR
    lDefault : t_charge_qualifier := cChargeQualifierNone;
    lValue : t_charge_qualifier := cChargeQualifierNone;
    lPending : t_charge_qualifier := cChargeQualifierNone;
  END_VAR

            
          

METHOD operator
  VAR_INPUT
    override : BOOL;
  END_VAR
                  IF (override) THEN
	lValue := Default;
ELSE
	lValue := lPending;
END_IF

lPending := Default;

                
END_METHOD

PROPERTY Default : t_charge_qualifier
GET
                    Default := lDefault;
                  
END_GET
SET
                    lDefault := Default;

                  
END_SET
END_PROPERTY

PROPERTY Pending : t_charge_qualifier
GET
                    Pending := lPending;
                  
END_GET
SET
                    IF (Pending=cChargeQualifierNone) THEN
	RETURN;
END_IF

IF (((lPending=cChargeQualifierCharge) AND
	(Pending=cChargeQualifierDischarge)) OR
	((lPending=cChargeQualifierDischarge) AND
	(Pending=cChargeQualifierCharge))) THEN
	lPending := cChargeQualifierBoth;
	RETURN;
END_IF

lPending := MIN(lPending,Pending);


                  
END_SET
END_PROPERTY

PROPERTY Value : t_charge_qualifier
GET
                    Value := lValue;
                  
END_GET
END_PROPERTY
END_FUNCTION_BLOCK

FUNCTION_BLOCK PendingInterlockState
  VAR
    lDefault : t_interlock_state := cInterlockStateGood;
    lValue : t_interlock_state := cInterlockStateGood;
    lPending : t_interlock_state := cInterlockStateGood;
  END_VAR

            
          

METHOD operator
  VAR_INPUT
    override : BOOL;
  END_VAR
                  IF (override) THEN
	lValue := Default;
ELSE
	lValue := lPending;
END_IF

lPending := Default;

                
END_METHOD

PROPERTY Default : t_interlock_state
GET
                    Default := lDefault;
                  
END_GET
SET
                    lDefault := Default;

                  
END_SET
END_PROPERTY

PROPERTY Pending : t_interlock_state
GET
                    Pending := lPending;
                  
END_GET
SET
                    IF (Pending=cInterlockStateNone) THEN
	RETURN;
END_IF

IF (((lPending=cInterlockStateErrorNegative) AND
	(Pending=cInterlockStateErrorPositive)) OR
	((lPending=cInterlockStateErrorPositive) AND
	(Pending=cInterlockStateErrorNegative))) THEN
	lPending := cInterlockStateError;
	RETURN;
END_IF

lPending := MIN(lPending,Pending);

                  
END_SET
END_PROPERTY

PROPERTY Value : t_interlock_state
GET
                    Value := lValue;
                  
END_GET
END_PROPERTY
END_FUNCTION_BLOCK

FUNCTION_BLOCK PendingPercentage
  VAR
    lDefault : t_percentage := 1.0;
    lValue : t_percentage := 1.0;
    lPending : t_percentage := 1.0;
  END_VAR

            
          

METHOD operator
  VAR_INPUT
    override : BOOL;
  END_VAR
                  IF (override) THEN
	lValue :=Default;
ELSE
	lValue := lPending;
END_IF

lPending := Default;

                
END_METHOD

PROPERTY Default : t_percentage
GET
                    Default := lDefault;
                  
END_GET
SET
                    lDefault := Default;

                  
END_SET
END_PROPERTY

PROPERTY Pending : t_percentage
GET
                    Pending := lPending;
                  
END_GET
SET
                    lPending := MIN(lPending,ABS(Pending));

                  
END_SET
END_PROPERTY

PROPERTY Value : t_percentage
GET
                    Value := lValue;
                  
END_GET
END_PROPERTY
END_FUNCTION_BLOCK

FUNCTION_BLOCK PendingSystemControl
  VAR
    lDefault : t_system_control := cSystemControlNone;
    lValue : t_system_control := cSystemControlNone;
    lPending : t_system_control := cSystemControlNone;
  END_VAR

            
          

METHOD operator
  VAR_INPUT
    override : BOOL;
  END_VAR
                  IF (override) THEN
	lValue := Default;
ELSE
	lValue := lPending;
END_IF

lPending := Default;

                
END_METHOD

PROPERTY Default : t_system_control
GET
                    Default := lDefault;
                  
END_GET
SET
                    lDefault := Default;

                  
END_SET
END_PROPERTY

PROPERTY Pending : t_system_control
GET
                    Pending := lPending;
                  
END_GET
SET
                    lPending := MIN(lPending,Pending);

                  
END_SET
END_PROPERTY

PROPERTY Value : t_system_control
GET
                    Value := lValue;
                  
END_GET
END_PROPERTY
END_FUNCTION_BLOCK

FUNCTION_BLOCK PendingSystemStateDown
  VAR
    lDefault : t_system_state := cSystemStateInitialized;
    lValue : t_system_state := cSystemStateInitialized;
    lPending : t_system_state := cSystemStateInitialized;
  END_VAR

            
          

METHOD operator
  VAR_INPUT
    override : BOOL;
  END_VAR
                  IF (override) THEN
	lValue := Default;
ELSE
	lValue := lPending;
END_IF

lPending := Default;


                
END_METHOD

PROPERTY Default : t_system_state
GET
                    Default := lDefault;
                  
END_GET
SET
                    lDefault := Default;

                  
END_SET
END_PROPERTY

PROPERTY Pending : t_system_state
GET
                    Pending := lPending;
                  
END_GET
SET
                    IF (Pending=cSystemStateNone) THEN
	RETURN;
END_IF

lPending := MAX(lPending,Pending);

                  
END_SET
END_PROPERTY

PROPERTY Value : t_system_state
GET
                    Value := lValue;
                  
END_GET
END_PROPERTY
END_FUNCTION_BLOCK

FUNCTION_BLOCK PendingSystemStateUp
  VAR
    lDefault : t_system_state := cSystemStateOperational;
    lValue : t_system_state := cSystemStateOperational;
    lPending : t_system_state := cSystemStateOperational;
  END_VAR

            
          

METHOD operator
  VAR_INPUT
    override : BOOL;
  END_VAR
                  IF (override) THEN
	lValue := Default;
ELSE
	lValue := lPending;
END_IF

lPending := Default;

                
END_METHOD

PROPERTY Default : t_system_state
GET
                    Default := lDefault;
                  
END_GET
SET
                    lDefault := Default;

                  
END_SET
END_PROPERTY

PROPERTY Pending : t_system_state
GET
                    Pending := lPending;
                  
END_GET
SET
                    IF (Pending=cSystemStateNone) THEN
	RETURN;
END_IF

lPending := MIN(lPending,Pending);

                  
END_SET
END_PROPERTY

PROPERTY Value : t_system_state
GET
                    Value := lValue;
                  
END_GET
END_PROPERTY
END_FUNCTION_BLOCK

FUNCTION_BLOCK Reportable EXTENDS NonOperationalParticleSet
  VAR
    lVROverride : ValueReferenceBool;
    lOverride : BOOL := FALSE;
    lVRSuppress : ValueReferenceBool;
    lSuppress : BOOL := TRUE;
    lVRSuppressAfterCountDown : ValueReferenceBool;
    lSuppressAfterCountDown : BOOL := FALSE;
    lVRSupressCountDown : ValueReferenceUINT;
    lSupressCountDown : UINT := 0;
    lVRChannelMask : ValueReferenceUINT;
    lChannelMask : UINT := 0;
    lResolvedSuppressAfterCountDown : BOOL := FALSE;
    lReportedTimeStep : t_timestep;
    lReportedCount : UDINT := 0;
    lPropagateCount : USINT := 0;
  END_VAR

            
          

METHOD _report
                  lReportedCount := lReportedCount + 1;
lReportedTimeStep := gSystemServices.Cycle.TimeStep;
                
END_METHOD

METHOD describe
  VAR_INPUT
    executeContext : POINTER TO ExecuteContext;
  END_VAR
  VAR
    str : t_stream_string;
  END_VAR
                  SUPER^.describe(executeContext);

IF (executeContext^.matchOption(cExecuteOptionSyntax)) THEN
	executeContext^.describeSyntaxExecutable(sCommandChannelMaskAdd);
	executeContext^.describeSyntaxExecutable(sCommandChannelMaskDelete);
	executeContext^.describeSyntaxExecutable(sCommandChannelMaskClear);

	RETURN;
END_IF

IF (executeContext^.matchOption(cExecuteOptionParameter)) THEN	
	RETURN;
END_IF

executeContext^.appendPair('Override',gTypeHandler.getTokenForUSINT(BOOL_TO_USINT(Override)),FALSE,TRUE);
executeContext^.appendPair('Suppress',gTypeHandler.getTokenForUSINT(BOOL_TO_USINT(Suppress)),FALSE,TRUE);

IF (executeContext^.matchOption(cExecuteOptionSyntax)) THEN	
	executeContext^.appendPair('reported',gTypeHandler.getTokenForUDINT(ReportedCount),FALSE,TRUE);
END_IF

                
END_METHOD

METHOD initialize
                  lVROverride.initializeValueReference(lOverride,NopSelf,'Override','Prevent any activation','',cValueStyleParameter);
lVRSuppress.initializeValueReference(lSuppress,NopSelf,'Suppress','Suppress notification','',cValueStyleConfigurable);
lVRSuppressAfterCountDown.initializeValueReference(lSuppressAfterCountDown,NopSelf,'SuppressAfter','Suppress after count down ends','',cValueStyleConfigurable);
lVRSupressCountDown.initializeValueReference(lSupressCountDown,NopSelf,'SuppressCntdwn','Count down length','timestep',cValueStyleConfigurable);
lVRChannelMask.initializeValueReference(lChannelMask,NopSelf,'ChannelMask','Channel notification mask','',cValueStyleParameter);

lReportedCount := 0;
lChannelMask := 0;

SUPER^.initialize();

                
END_METHOD

METHOD propagate
                  lPropagateCount := lPropagateCount + 1;

                
END_METHOD

METHOD report
  VAR_INPUT
    override : BOOL;
  END_VAR
                  IF ((override) OR 
	(Override)) THEN
	RETURN;
END_IF

_report();

IF (lSuppressAfterCountDown) THEN
	IF (lSupressCountDown>0) THEN
		lResolvedSuppressAfterCountDown := FALSE;
		lSupressCountDown := lSupressCountDown - 1;
	ELSE
		lResolvedSuppressAfterCountDown := TRUE;
	END_IF
END_IF

                
END_METHOD

METHOD execute
  VAR_INPUT
    executeContext : POINTER TO ExecuteContext;
  END_VAR
  VAR
    token : t_token_string;
    mask : t_channel_mask;
  END_VAR
                  IF (executeContext=0) THEN
	RETURN;
END_IF

IF (executeContext^.matchCommand(sCommandChannelMaskAdd)) THEN
	
	IF (NOT(executeContext^.configureEnum(cEnumTypeChannelMask,cTokenFeature,mask,TRUE,THIS))) THEN
		RETURN;
	END_IF
	
	lChannelMask := lChannelMask OR INT_TO_UINT(mask);
	RETURN;
END_IF

IF (executeContext^.matchCommand(sCommandChannelMaskDelete)) THEN

	IF (NOT(executeContext^.configureEnum(cEnumTypeChannelMask,cTokenFeature,mask,TRUE,THIS))) THEN
		RETURN;
	END_IF
	
	lChannelMask := lChannelMask AND NOT(INT_TO_UINT(mask));
	RETURN;
END_IF

IF (executeContext^.matchCommand(sCommandChannelMaskClear)) THEN	
	lChannelMask := 0;
	RETURN;
END_IF

SUPER^.execute(executeContext);

                
END_METHOD

METHOD trigger
  VAR_INPUT
    override : BOOL;
  END_VAR
                  IF (override) THEN
	RETURN;
END_IF 

report(FALSE);
                
END_METHOD

PROPERTY ChannelMask : UINT
GET
                    ChannelMask := lChannelMask;
                  
END_GET
SET
                    lChannelMask := ChannelMask;
                  
END_SET
END_PROPERTY

PROPERTY Override : BOOL
GET
                    Override := lOverride;
                  
END_GET
SET
                    lOverride := Override;
                  
END_SET
END_PROPERTY

PROPERTY ReportedCount : UDINT
GET
                    ReportedCount := lReportedCount;
                  
END_GET
END_PROPERTY

PROPERTY ReportedTimeStep : t_timestep
GET
                    ReportedTimeStep := lReportedTimeStep;
                  
END_GET
SET
                    lReportedTimeStep := ReportedTimeStep;
                  
END_SET
END_PROPERTY

PROPERTY ResolvedSuppress : BOOL
GET
                    ResolvedSuppress := ((lSuppress) OR
	(lResolvedSuppressAfterCountDown));

                  
END_GET
END_PROPERTY

PROPERTY Suppress : BOOL
GET
                    Suppress := lSuppress;
                  
